	Version history:
	Date        | Version   | Author                    | Remark
	----------------------------------------------------------------------------------------
	 30/03/2023 | 0.1       | R.Golonka                 | First release TIA 17.0 | DHL Munich
	 18/08/2023 | 2.0       | Stefanos Theocharis       | align with Parma UDT
	 06/09/2023 | 2.1       | M.Diebel                  | Reset energy save when NewObjectID is created
	 13/03/2024 | 2.2      | S. Nieswiec                | Added to new baseline

	 *)

	REGION 1 - Chute status move

	    #s_UDT_Downstream_Sorter.Full := #i_UDT_Outfeed2StatesStatus.Specific.ChuteFull;// Downstream sorter status full update

	    #s_UDT_Downstream_Sorter.HalfFull := #i_UDT_Outfeed2StatesStatus.Specific.ChuteHalfFull;   // Downstream sorter status half-full update

	END_REGION

	REGION 2 - Send ready to recevie to crossbelt

	    // Set ready to recevie to Xbelt (when Chute is RTR then XBelt can discharge)
	    #s_UDT_Downstream_Sorter.ReadyToReceive := #iq_UDT_ChuteExternalHandshake.RTR AND (#i_UDT_AssociatedConveyorInterface.VFDatSpeed OR NOT #ix_ConfigHorizontalOutfeed);

	END_REGION

	REGION 3 - Downstream Sorter

	    // Downstream sorter functionality when horizontal outfeed mode is active
	    IF #ix_ConfigHorizontalOutfeed THEN
	        #s_UDT_Downstream_Sorter.Running := #i_UDT_AssociatedConveyorInterface.RunFwd AND NOT #i_UDT_AssociatedConveyorInterface.ManualModeActive;

	    ELSE
	        #s_UDT_Downstream_Sorter.Running := #iq_UDT_ChuteExternalHandshake.RTR; // Downstream sorter functionality when spiral mode is active

	    END_IF;

	END_REGION

	REGION 4 - Package update

	    // Move the current ID to position 0
	    #sa_ExchangeObjectID[0] := #i_UDT_Sorter_Downstream.DischargedObjectID;

	    // When the ID is different with previous ID do:
	    IF #sa_ExchangeObjectID[0] <> #sa_ExchangeObjectID[1] THEN
	        // Update new object
	        #s_UDT_XBeltExitInterface.NewObjectID := TRUE;
	        // Update obejct ID
	        #s_UDT_XBeltExitInterface.ObjectID := #i_UDT_Sorter_Downstream.DischargedObjectID;
	        // Update product lenght
	        #s_UDT_XBeltExitInterface.ProductLength := DINT_TO_INT(#i_UDT_Sorter_Downstream.DischargedPackageLength MOD #c_MaximumLength);
	        // Setting actual value to previous one
	        #sa_ExchangeObjectID[1] := #sa_ExchangeObjectID[0];
	    ELSE
	        #s_UDT_XBeltExitInterface.NewObjectID := FALSE;
	    END_IF;

	    #iq_UDT_ChuteExternalHandshake.RTS := #s_UDT_XBeltExitInterface.NewObjectID;    // Conveyor ready to send if parcel diverted
	    #iq_UDT_ChuteExternalHandshake.ResetEnergySave := #s_UDT_XBeltExitInterface.NewObjectID;
	END_REGION

	REGION 5 - Output update

	    #q_UDT_Downstream_Sorter := #s_UDT_Downstream_Sorter;    // Move UDT Downstream Sorter to output

	    #q_UDT_XBeltExitInterface := #s_UDT_XBeltExitInterface;    // Move Xbelt Exit interface

	END_REGION

	REGION 6 - Status

	    #s_UDT_XBeltExitStatus.ChuteDisabled := #i_UDT_Sorter_Downstream.Basic.ChuteDisabled;   // Status HMI upadate chute disabled

	    #s_UDT_XBeltExitStatus.ChuteJam := #i_UDT_Sorter_Downstream.Basic.ChuteJam;   // Status HMI upadate chute jammed

	    #s_UDT_XBeltExitStatus.ChuteSensorIncongruence := #i_UDT_Sorter_Downstream.Basic.ChuteSensorIncongruence;    // Status HMI update chute sensor incongrunce

	    #q_UDT_XBeltExitStatus := #s_UDT_XBeltExitStatus;  // Move status static to output

	END_REGION


END_FUNCTION_BLOCK

FUNCTION_BLOCK "FB_VFD_MultiControl_Universal_Full"
{ S7_Optimized_Access := 'TRUE' }
AUTHOR : 'KBA-PM'
VERSION : 0.1
// ATTRIBUTES
// AUTO_NUMBER = True
// BLOCK_NUMBER = 106
// END_ATTRIBUTES
   VAR_INPUT
      i_UDT_VFDConfiguration { ExternalAccessible := 'False'; ExternalVisible := 'False'; ExternalWritable := 'False'} : "UDT_VFD_MultiControl_Configuration";   //   VFD configuration structure
      i_UDT_VFDInputs { ExternalAccessible := 'False'; ExternalVisible := 'False'; ExternalWritable := 'False'} : "UDT_VFD_MultiControl_Universal_Full";   //   VFD inputs structure
      ii_MotorNumber { ExternalAccessible := 'False'; ExternalVisible := 'False'; ExternalWritable := 'False'} : Int;   //   Motor number that is connected to the Multicontrol module [1,2,3 or 4]
      ix_PowerOK { ExternalAccessible := 'False'; ExternalVisible := 'False'; ExternalWritable := 'False'} : Bool;   //   TRUE when External Power OK
      ix_SafetyOK { ExternalAccessible := 'False'; ExternalVisible := 'False'; ExternalWritable := 'False'} : Bool;   //   TRUE when Safety OK
      ix_SimulationModeActive { ExternalAccessible := 'False'; ExternalVisible := 'False'; ExternalWritable := 'False'} : Bool;   //   TRUE when Simulation mode active
   END_VAR

   VAR_OUTPUT
      q_UDT_HMIStatus { ExternalAccessible := 'False'; ExternalVisible := 'False'; ExternalWritable := 'False'} : "UDT_VfdStatus";   //   HMI status structure
      qsi_UDT_VFDSpeed { ExternalAccessible := 'False'; ExternalVisible := 'False'; ExternalWritable := 'False'} : SInt;   //   VFD speed setpoint
   END_VAR

   VAR_IN_OUT
      iq_UDT_ConveyorInterface : "UDT_ConveyorInterface";   //   Conveyor interface structure
      iq_UDT_VFDStatistics : "UDT_VfdStatistics";   //   Statistics structure
   END_VAR

   VAR
      s_FB_TimerOnOffDelayCheckSupply { ExternalAccessible := 'False'; ExternalVisible := 'False'; ExternalWritable := 'False'; S7_SetPoint := 'False'} : "FB_TimerOnOffDelay";   //  "TimerOnOffDelay" - to delay time for VFD supply contactor
      s_FB_TimerOnOffDelay_ProfinetNotOnlineMasking { ExternalAccessible := 'False'; ExternalVisible := 'False'; ExternalWritable := 'False'; S7_SetPoint := 'False'} : "FB_TimerOnOffDelay";   //   "TimerOnOffDelay" - to delay time for profinet not online masking
      s_FB_TimerOnOffDelay_ProfinetSlaveErrorMasking { ExternalAccessible := 'False'; ExternalVisible := 'False'; ExternalWritable := 'False'; S7_SetPoint := 'False'} : "FB_TimerOnOffDelay";   //   "TimerOnOffDelay" - to delay time for profinet error masking
      s_FB_TimerOnOffDelay_Instance { ExternalAccessible := 'False'; ExternalVisible := 'False'; ExternalWritable := 'False'; S7_SetPoint := 'False'} : "FB_TimerOnOffDelay";   //   "TimerOnOffDelay" - to delay time for Instance
      s_FB_TimerOnOffDelay_SafetyOK { ExternalAccessible := 'False'; ExternalVisible := 'False'; ExternalWritable := 'False'; S7_SetPoint := 'False'} : "FB_TimerOnOffDelay";   //   "TimerOnOffDelay" - to delay time for safety
      s_FB_TimerOnOffDelay_RunCommand { ExternalAccessible := 'False'; ExternalVisible := 'False'; ExternalWritable := 'False'; S7_SetPoint := 'False'} : "FB_TimerOnOffDelay";   //   "TimerOnOffDelay" - to delay time for run command motor
      s_R_TRIG_RunForward {InstructionName := 'R_TRIG'; LibVersion := '1.0'; ExternalAccessible := 'False'; ExternalVisible := 'False'; ExternalWritable := 'False'; S7_SetPoint := 'False'} : R_TRIG;   //   Rising edge of Run forward signal
      s_R_TRIG_RunReverse {InstructionName := 'R_TRIG'; LibVersion := '1.0'; ExternalAccessible := 'False'; ExternalVisible := 'False'; ExternalWritable := 'False'; S7_SetPoint := 'False'} : R_TRIG;   //   Rising edge of Run reverse
      s_R_TRIG_PNSlaveNotOnline {InstructionName := 'R_TRIG'; LibVersion := '1.0'; ExternalAccessible := 'False'; ExternalVisible := 'False'; ExternalWritable := 'False'; S7_SetPoint := 'False'} : R_TRIG;   //   Rising edge for trigger Profinet slave not online statistics
      s_R_TRIG_PNSlaveError {InstructionName := 'R_TRIG'; LibVersion := '1.0'; ExternalAccessible := 'False'; ExternalVisible := 'False'; ExternalWritable := 'False'; S7_SetPoint := 'False'} : R_TRIG;   //   Rising edge for trigger Profinet slave error statistics
      s_R_TRIG_InternalError {InstructionName := 'R_TRIG'; LibVersion := '1.0'; ExternalAccessible := 'False'; ExternalVisible := 'False'; ExternalWritable := 'False'; S7_SetPoint := 'False'} : R_TRIG;   //   Rising edge for trigger Internal VFD Error statistics
      s_R_TRIG_Running {InstructionName := 'R_TRIG'; LibVersion := '1.0'; ExternalAccessible := 'False'; ExternalVisible := 'False'; ExternalWritable := 'False'; S7_SetPoint := 'False'} : R_TRIG;   //   Rising edge for starting of the running signal
      s_R_TRIG_Instance {InstructionName := 'R_TRIG'; LibVersion := '1.0'; ExternalAccessible := 'False'; ExternalVisible := 'False'; ExternalWritable := 'False'; S7_SetPoint := 'False'} : R_TRIG;   //   Raising edge for Instance
      s_R_TRIG_NewPNSlaveError {InstructionName := 'R_TRIG'; LibVersion := '1.0'; ExternalAccessible := 'False'; ExternalVisible := 'False'; ExternalWritable := 'False'; S7_SetPoint := 'False'} : R_TRIG;   //   New profinet slave error trigger
      s_R_TRIG_NewPNSlaveNotOnline {InstructionName := 'R_TRIG'; LibVersion := '1.0'; ExternalAccessible := 'False'; ExternalVisible := 'False'; ExternalWritable := 'False'; S7_SetPoint := 'False'} : R_TRIG;   //   New profinet slave not online trigger
      s_UDT_HMIStatus { ExternalAccessible := 'False'; ExternalVisible := 'False'; ExternalWritable := 'False'; S7_SetPoint := 'False'} : "UDT_VfdStatus";   //   HMI status structure
      s_UDT_PNDevice { ExternalAccessible := 'False'; ExternalVisible := 'False'; ExternalWritable := 'False'; S7_SetPoint := 'False'} : "UDT_PNDevice";   //   PN device info structure
      ss_VFDGeoStruct {InstructionName := 'GEOADDR'; LibVersion := '1.0'; ExternalAccessible := 'False'; ExternalVisible := 'False'; ExternalWritable := 'False'; S7_SetPoint := 'False'} : GEOADDR;   //   Geo structure indicate to telegram
      ss_RDREC { ExternalAccessible := 'False'; ExternalVisible := 'False'; ExternalWritable := 'False'} : Struct   //   Read error code record structure
         Valid { ExternalAccessible := 'False'; ExternalVisible := 'False'; ExternalWritable := 'False'} : Bool;   //      Read operation is done
         Busy { ExternalAccessible := 'False'; ExternalVisible := 'False'; ExternalWritable := 'False'} : Bool;   //      Read operation is in progress
         Error { ExternalAccessible := 'False'; ExternalVisible := 'False'; ExternalWritable := 'False'} : Bool;   //      Read operation has an error
         Status { ExternalAccessible := 'False'; ExternalVisible := 'False'; ExternalWritable := 'False'} : DWord;   //      Read operation status
         Lenght { ExternalAccessible := 'False'; ExternalVisible := 'False'; ExternalWritable := 'False'} : UInt;   //      Lenght of the read record
      END_STRUCT;
      ss_WRREC { ExternalAccessible := 'False'; ExternalVisible := 'False'; ExternalWritable := 'False'} : Struct   //   Write record structure
         Acceleration { ExternalAccessible := 'False'; ExternalVisible := 'False'; ExternalWritable := 'False'} : Struct   //      Acceleration
            REQ { ExternalAccessible := 'False'; ExternalVisible := 'False'; ExternalWritable := 'False'} : Bool;   //      Requirement
            Index { ExternalAccessible := 'False'; ExternalVisible := 'False'; ExternalWritable := 'False'} : DInt;   //      Index
            Done { ExternalAccessible := 'False'; ExternalVisible := 'False'; ExternalWritable := 'False'} : Bool;   //      Operation is done
            Busy { ExternalAccessible := 'False'; ExternalVisible := 'False'; ExternalWritable := 'False'} : Bool;   //      Write operation is in progress
            Error { ExternalAccessible := 'False'; ExternalVisible := 'False'; ExternalWritable := 'False'} : Bool;   //      Write operation has an error
            Status { ExternalAccessible := 'False'; ExternalVisible := 'False'; ExternalWritable := 'False'} : DWord;   //      Write operation status
            Data { ExternalAccessible := 'False'; ExternalVisible := 'False'; ExternalWritable := 'False'} : Word;   //      Data to write
         END_STRUCT;
         Deceleration { ExternalAccessible := 'False'; ExternalVisible := 'False'; ExternalWritable := 'False'} : Struct   //      Deceleration
            REQ { ExternalAccessible := 'False'; ExternalVisible := 'False'; ExternalWritable := 'False'} : Bool;   //      Requirement
            Index { ExternalAccessible := 'False'; ExternalVisible := 'False'; ExternalWritable := 'False'} : DInt;   //      Index
            Done { ExternalAccessible := 'False'; ExternalVisible := 'False'; ExternalWritable := 'False'} : Bool;   //      Operation is done
            Busy { ExternalAccessible := 'False'; ExternalVisible := 'False'; ExternalWritable := 'False'} : Bool;   //      Write operation is in progress
            Error { ExternalAccessible := 'False'; ExternalVisible := 'False'; ExternalWritable := 'False'} : Bool;   //      Write operation has an error
            Status { ExternalAccessible := 'False'; ExternalVisible := 'False'; ExternalWritable := 'False'} : DWord;   //      Write operation status
            Data { ExternalAccessible := 'False'; ExternalVisible := 'False'; ExternalWritable := 'False'} : Word;   //      Data to write
         END_STRUCT;
      END_STRUCT;
      s_RDREC_ErrorCode {InstructionName := 'RDREC'; LibVersion := '1.0'; ExternalAccessible := 'False'; ExternalVisible := 'False'; ExternalWritable := 'False'; S7_SetPoint := 'False'} : RDREC;   //   Read error code record instruction
      s_WRREC_ACC {InstructionName := 'WRREC'; LibVersion := '1.1'; ExternalAccessible := 'False'; ExternalVisible := 'False'; ExternalWritable := 'False'; S7_SetPoint := 'False'} : WRREC;   //   Write acceleration record inctruction
      s_WRREC_DEC {InstructionName := 'WRREC'; LibVersion := '1.1'; ExternalAccessible := 'False'; ExternalVisible := 'False'; ExternalWritable := 'False'; S7_SetPoint := 'False'} : WRREC;   //   Write deceleration record instruction
      shw_VFD_Telegram { ExternalAccessible := 'False'; ExternalVisible := 'False'; ExternalWritable := 'False'} : HW_ANY;   //   Free telegram's HW_ID
      sr_MaximumSpeed { ExternalAccessible := 'False'; ExternalVisible := 'False'; ExternalWritable := 'False'} : Real;   //   Maximum speed [mm/s]
      sr_SpeedsetpointCorrected { ExternalAccessible := 'False'; ExternalVisible := 'False'; ExternalWritable := 'False'} : Real;   //  Speedsetpoint corrected with factor
      sw_ErrorCode { ExternalAccessible := 'False'; ExternalVisible := 'False'; ExternalWritable := 'False'} : Word;   //   VFD error code
      si_RequiredSpeedSetpoint { ExternalAccessible := 'False'; ExternalVisible := 'False'; ExternalWritable := 'False'} : Int;   //   Required speed setpoint
      si_AccelerationSetpoint { ExternalAccessible := 'False'; ExternalVisible := 'False'; ExternalWritable := 'False'} : Int;   //   Acceleration setpoint value
      si_DecelerationSetpoint { ExternalAccessible := 'False'; ExternalVisible := 'False'; ExternalWritable := 'False'} : Int;   //   Deceleration setpoint value
      si_AccelerationOld { ExternalAccessible := 'False'; ExternalVisible := 'False'; ExternalWritable := 'False'} : Int;   //   Old acceleration value
      si_DecelerationOld { ExternalAccessible := 'False'; ExternalVisible := 'False'; ExternalWritable := 'False'} : Int;   //   Old deceleration value
      si_ActualSpeed { ExternalAccessible := 'False'; ExternalVisible := 'False'; ExternalWritable := 'False'} : Int;   //   Actual speed in [mm/s]
      si_Log2GeoReturn { ExternalAccessible := 'False'; ExternalVisible := 'False'; ExternalWritable := 'False'} : Int;   //   Log2Geo function return
      si_Geo2LogReturn { ExternalAccessible := 'False'; ExternalVisible := 'False'; ExternalWritable := 'False'} : Int;   //   Geo2Log function return
      sx_PNSlaveErrorCount { ExternalAccessible := 'False'; ExternalVisible := 'False'; ExternalWritable := 'False'} : Int;   //   Profinet slave error counter
      sx_PNSlaveNotOnlineCount { ExternalAccessible := 'False'; ExternalVisible := 'False'; ExternalWritable := 'False'} : Int;   //   Profinet slave not online counter
      ssi_MotorSpeed { ExternalAccessible := 'False'; ExternalVisible := 'False'; ExternalWritable := 'False'} : SInt;   //   Motor speed value
      sx_ConfigurationError { ExternalAccessible := 'False'; ExternalVisible := 'False'; ExternalWritable := 'False'} : Bool;   //   Commissioning: configuration error
      sx_PNDeviceHealthy { ExternalAccessible := 'False'; ExternalVisible := 'False'; ExternalWritable := 'False'} : Bool;   //   Profinet device is online and error free
      sx_PowerOk { ExternalAccessible := 'False'; ExternalVisible := 'False'; ExternalWritable := 'False'} : Bool;   //   Communication, safety and power are available
      sx_VFD_Available { ExternalAccessible := 'False'; ExternalVisible := 'False'; ExternalWritable := 'False'} : Bool;   //   Hardware of VFD is ok
      sx_ErrorActive { ExternalAccessible := 'False'; ExternalVisible := 'False'; ExternalWritable := 'False'} : Bool;   //   Block has an error
      sx_InvalidMotorNumber { ExternalAccessible := 'False'; ExternalVisible := 'False'; ExternalWritable := 'False'} : Bool;   //   Invalid motor error
      sx_MotorError { ExternalAccessible := 'False'; ExternalVisible := 'False'; ExternalWritable := 'False'} : Bool;   //   Motor error
      sx_EnableOperation { ExternalAccessible := 'False'; ExternalVisible := 'False'; ExternalWritable := 'False'} : Bool;   //   Enable operation signal
      sx_RunVFDForward { ExternalAccessible := 'False'; ExternalVisible := 'False'; ExternalWritable := 'False'} : Bool;   //   Start VFD forward
      sx_RunVFDReverse { ExternalAccessible := 'False'; ExternalVisible := 'False'; ExternalWritable := 'False'} : Bool;   //   Start VFD backward
      sx_AccelerationDone { ExternalAccessible := 'False'; ExternalVisible := 'False'; ExternalWritable := 'False'} : Bool;   //   Acceleration is written
      sx_DecelerationDone { ExternalAccessible := 'False'; ExternalVisible := 'False'; ExternalWritable := 'False'} : Bool;   //   Deceleration is written
      sx_SpeedSetpointReached { ExternalAccessible := 'False'; ExternalVisible := 'False'; ExternalWritable := 'False'} : Bool;   //   Motor is running at requested speed
      sx_ErrorDone { ExternalAccessible := 'False'; ExternalVisible := 'False'; ExternalWritable := 'False'} : Bool;   //   Error code is read
      sx_SafetyOK { ExternalAccessible := 'False'; ExternalVisible := 'False'; ExternalWritable := 'False'} : Bool;   //   Safety ok
      sx_MaskingReset { ExternalAccessible := 'False'; ExternalVisible := 'False'; ExternalWritable := 'False'} : Bool;   //   Masking reset
      sx_PNSlaveError { ExternalAccessible := 'False'; ExternalVisible := 'False'; ExternalWritable := 'False'} : Bool;   //   Profinet slave error
      sx_PNSlaveNotOnline { ExternalAccessible := 'False'; ExternalVisible := 'False'; ExternalWritable := 'False'} : Bool;   //   Profinet slave not online
      s_R_TRIG_PNSlaveNotOnline_Acyclic {InstructionName := 'R_TRIG'; LibVersion := '1.0'; ExternalAccessible := 'False'; ExternalVisible := 'False'; ExternalWritable := 'False'; S7_SetPoint := 'False'} : R_TRIG;
   END_VAR

   VAR CONSTANT
      ci_VFDArea : UInt := 1;   //   Area ID of IO Profinet devices
      ci_SubmoduleHWType : UInt := 5;   //   Submodule HW_type number
      ci_TelegramSlot : UInt := 2;   //   Free Siemens telegram slot
      ci_TelegramSubslot : UInt := 1;   //   Free Siemens telegram subslot
      cdi_ErrorCodeIndex : DInt := 17154;   //   Error code index
      cdi_AccelerationIndex : DInt := 18200;   //   Acceleration index
      cdi_DecelerationIndex : DInt := 18204;   //   Deceleration index
   END_VAR


BEGIN
	(*
	----------------------------------------------------------------------------------------
	|                                                                                      |
	|  Copyright  2023             FORTNA Europe BV                                        |
	|  All Rights Reserved         Netherlands                                             |
	|                                                                                      |
	----------------------------------------------------------------------------------------

	Version history:
	Date        | Version   | Author        | Remark
	----------------------------------------------------------------------------------------
	08/11/2019  | 3.0       | A. Nowak      | Initial version
	18/03/2020  | 3.1       | K.Pokorski    | Adapting reviews
	10/06/2021  | 3.2       | L.Klar        | Region 9.1 - #ssi_MotorSpeed = 0 condition commented
	17/11/2021  | 3.3       | P.Gryszczyk   | Region 2 - RunCommand timer changed conditions
	18/02/2021  | 3.4       | P.Gryszczyk   | Region 4 - PNNotOnline and PNSlaveError masking, sending reset to system
	24/05/2023  | 3.5       | S.Nikodem     | Update to DHL Munich specification
	04/07/2023  | 3.7       | P.Gryszczyk   | Changed the PNSlaveNotOnline to R_TRIG for the acyclic writing logic
	13/03/2024  | 4.1       | S. Nieswiec   | Added to new baseline
	*)

	REGION 1 - Get Device Profinet number

	    // Getting information about Profinet Device.
	    "FC_GetDevicePN"(is_PNDeviceName := #i_UDT_VFDConfiguration.VFDPNDeviceName,
	                     ix_SimulationModeActive := #ix_SimulationModeActive,
	                     iqUDT_PND := #s_UDT_PNDevice);

	END_REGION

	REGION 2 - Motor number validation

	    // Check the motor number and copy the it's error status and speed.
	    CASE (#ii_MotorNumber)
	    OF
	        1:
	            // Delay
	            #s_FB_TimerOnOffDelay_RunCommand(iudi_OnDelayTime := 1500,
	                                             ix_SignalToDelay :=
	                                             (#sx_RunVFDForward
	                                             OR #sx_RunVFDReverse)
	                                             AND #i_UDT_VFDInputs.CurrentMotor1 < #i_UDT_VFDConfiguration.MinimumCurrentWhenRunninng);

	            #ssi_MotorSpeed := #i_UDT_VFDInputs.SpeedMotor1;

	            IF (#s_FB_TimerOnOffDelay_RunCommand.qx_DelayedSignal AND #sx_EnableOperation) OR #i_UDT_VFDInputs.ErrorMotor1
	            THEN

	                #sx_MotorError := TRUE;

	            END_IF;
	        2:
	            #s_FB_TimerOnOffDelay_RunCommand(iudi_OnDelayTime := 1500,
	                                             ix_SignalToDelay :=
	                                             (#sx_RunVFDForward
	                                             OR #sx_RunVFDReverse)
	                                             AND #i_UDT_VFDInputs.CurrentMotor2 < #i_UDT_VFDConfiguration.MinimumCurrentWhenRunninng);

	            #ssi_MotorSpeed := #i_UDT_VFDInputs.SpeedMotor2;

	            IF (#s_FB_TimerOnOffDelay_RunCommand.qx_DelayedSignal AND #sx_EnableOperation) OR #i_UDT_VFDInputs.ErrorMotor2

	            THEN

	                #sx_MotorError := TRUE;

	            END_IF;
	        3:
	            #s_FB_TimerOnOffDelay_RunCommand(iudi_OnDelayTime := 1500,
	                                             ix_SignalToDelay :=
	                                             (#sx_RunVFDForward
	                                             OR #sx_RunVFDReverse)
	                                             AND #i_UDT_VFDInputs.CurrentMotor3 < #i_UDT_VFDConfiguration.MinimumCurrentWhenRunninng);

	            #ssi_MotorSpeed := #i_UDT_VFDInputs.SpeedMotor3;

	            IF (#s_FB_TimerOnOffDelay_RunCommand.qx_DelayedSignal AND #sx_EnableOperation) OR #i_UDT_VFDInputs.ErrorMotor3
	            THEN

	                #sx_MotorError := TRUE;

	            END_IF;
	        4:
	            #s_FB_TimerOnOffDelay_RunCommand(iudi_OnDelayTime := 1500,
	                                             ix_SignalToDelay :=
	                                             (#sx_RunVFDForward
	                                             OR #sx_RunVFDReverse)
	                                             AND #i_UDT_VFDInputs.CurrentMotor4 < #i_UDT_VFDConfiguration.MinimumCurrentWhenRunninng);

	            #ssi_MotorSpeed := #i_UDT_VFDInputs.SpeedMotor4;

	            IF (#s_FB_TimerOnOffDelay_RunCommand.qx_DelayedSignal AND #sx_EnableOperation) OR #i_UDT_VFDInputs.ErrorMotor4
	            THEN

	                #sx_MotorError := TRUE;

	            END_IF;

	        ELSE
	            #sx_InvalidMotorNumber := TRUE;
	    END_CASE;

	END_REGION

	REGION 3 - Reset errors

	    // Reset the errors on the command from the conveyor interface.
	    //
	    #s_R_TRIG_Instance(CLK := #ix_SafetyOK,
	                       Q => #sx_SafetyOK);

	    #s_FB_TimerOnOffDelay_Instance(iudi_OffDelayTime := 10000,
	                                   ix_SignalToDelay := #sx_SafetyOK,
	                                   qx_DelayedSignal => #sx_MaskingReset);


	    IF #iq_UDT_ConveyorInterface.InternalErrorReset THEN
	        #s_UDT_HMIStatus.PNSlaveNotonline := FALSE;
	        #s_UDT_HMIStatus.PNSlaveError := FALSE;
	        #s_UDT_HMIStatus.InternalError := FALSE;
	        #sx_InvalidMotorNumber := FALSE;
	        #sx_MotorError := FALSE;
	    END_IF;

	END_REGION

	REGION 4 - Hardware check

	    // Hardware will be available only after the delay, so the device has time for the initialization.
	    #s_FB_TimerOnOffDelayCheckSupply(iudi_OnDelayTime := 2000,
	                                     ix_SignalToDelay := #ix_PowerOK,
	                                     qx_DelayedSignal => #sx_PowerOk);

	    #s_FB_TimerOnOffDelay_ProfinetNotOnlineMasking(iudi_OnDelayTime := #i_UDT_VFDConfiguration.TimePNErrorMasking,
	                                                   iudi_OffDelayTime := 0,
	                                                   ix_SignalToDelay := #sx_PNSlaveNotOnline,
	                                                   qx_DelayedSignal => #s_UDT_HMIStatus.PNSlaveNotonline);

	    #s_FB_TimerOnOffDelay_ProfinetSlaveErrorMasking(iudi_OnDelayTime := #i_UDT_VFDConfiguration.TimePNErrorMasking,
	                                                    iudi_OffDelayTime := 0,
	                                                    ix_SignalToDelay := #sx_PNSlaveError,
	                                                    qx_DelayedSignal => #s_UDT_HMIStatus.PNSlaveError);

	    #s_R_TRIG_NewPNSlaveNotOnline(CLK := #sx_PNSlaveNotOnline);
	    #s_R_TRIG_NewPNSlaveError(CLK := #sx_PNSlaveError);
	    // Check if PN device is online.
	    IF NOT "DB_ProfinetDiagnostic".ProfinetNetworks[#s_UDT_PNDevice.PNNetworknumber].DeviceStatus[#s_UDT_PNDevice.PNDeviceNumber].DeviceState.Exist
	        AND NOT #ix_SimulationModeActive
	        AND #sx_PowerOk
	    THEN
	        #sx_PNSlaveNotOnline := TRUE;
	    ELSE
	        #sx_PNSlaveNotOnline := FALSE;
	    END_IF;

	    IF #s_R_TRIG_NewPNSlaveNotOnline.Q THEN
	        #sx_PNSlaveNotOnlineCount += 1;
	    END_IF;

	    // Check if PN device has an error.
	    IF "DB_ProfinetDiagnostic".ProfinetNetworks[#s_UDT_PNDevice.PNNetworknumber].DeviceStatus[#s_UDT_PNDevice.PNDeviceNumber].DeviceState.Error
	        AND NOT #ix_SimulationModeActive
	        AND #sx_PowerOk
	    THEN
	        #sx_PNSlaveError := TRUE;
	    ELSE
	        #sx_PNSlaveError := FALSE;
	    END_IF;

	    IF #s_R_TRIG_NewPNSlaveError.Q THEN
	        #sx_PNSlaveErrorCount += 1;
	    END_IF;

	    // Set bit when PN device is healthy (online and no error).
	    #sx_PNDeviceHealthy :=
	    NOT #s_UDT_HMIStatus.PNSlaveNotonline
	    AND NOT #s_UDT_HMIStatus.PNSlaveError
	    AND #s_UDT_PNDevice.PNDeviceFound
	    AND #sx_PowerOk;

	    // Set VFD available bit when all conditions are met.
	    #sx_VFD_Available :=
	    (NOT #sx_MotorError
	    AND #sx_PowerOk
	    AND #sx_PNDeviceHealthy)
	    OR #ix_SimulationModeActive;

	END_REGION

	REGION 5 - Extract telegram's HW_ID

	    // Extract telegram's HW_ID
	    #si_Log2GeoReturn := LOG2GEO(LADDR := "DB_ProfinetDiagnostic".ProfinetNetworks[#s_UDT_PNDevice.PNNetworknumber].DeviceStatus[#s_UDT_PNDevice.PNDeviceNumber].DeviceState.HW_ID, GEOADDR := #ss_VFDGeoStruct);
	    #ss_VFDGeoStruct.AREA := #ci_VFDArea;
	    #ss_VFDGeoStruct.HWTYPE := #ci_SubmoduleHWType;
	    #ss_VFDGeoStruct.STATION := INT_TO_UINT(#s_UDT_PNDevice.PNDeviceNumber);
	    #ss_VFDGeoStruct.SLOT := #ci_TelegramSlot;
	    #ss_VFDGeoStruct.SUBSLOT := #ci_TelegramSubslot;

	    #si_Geo2LogReturn := GEO2LOG(GEOADDR := #ss_VFDGeoStruct, LADDR => #shw_VFD_Telegram);

	END_REGION

	REGION 6 - Check errors

	    #s_FB_TimerOnOffDelay_SafetyOK(iudi_OnDelayTime := 10000,
	                                   ix_SignalToDelay := #ix_SafetyOK);

	    // Check if the motor has an error.
	    IF #s_FB_TimerOnOffDelay_SafetyOK.qx_DelayedSignal  //#ix_SafetyOK
	    THEN
	        #s_UDT_HMIStatus.InternalError := #sx_MotorError;

	    END_IF;
	    // Create trigger on error.
	    #s_R_TRIG_InternalError(CLK := #s_UDT_HMIStatus.InternalError);

	    // If the internal error occured, reset the error code read done signal.
	    IF #s_R_TRIG_InternalError.Q
	    THEN
	        #sx_ErrorDone := FALSE;
	    END_IF;

	    // If there is an internal error, read the error code from the Interroll VFD. Otherwise, reset it.
	    IF NOT #s_UDT_HMIStatus.InternalError
	    THEN
	        #s_UDT_HMIStatus.ErrorCode := 0;
	    ELSE
	        // Read the error code from the multicontrol.
	        #s_RDREC_ErrorCode(REQ := ((NOT #sx_ErrorDone OR "mx_FirstScan") AND NOT #s_UDT_HMIStatus.PNSlaveNotonline),
	                           ID := #shw_VFD_Telegram,
	                           INDEX := #cdi_ErrorCodeIndex,
	                           MLEN := 0,
	                           VALID => #ss_RDREC.Valid,
	                           BUSY => #ss_RDREC.Busy,
	                           ERROR => #ss_RDREC.Error,
	                           STATUS => #ss_RDREC.Status,
	                           LEN => #ss_RDREC.Lenght,
	                           RECORD := #sw_ErrorCode);

	        // IF error code is read, set the error code read signal and write it to the structure.
	        IF #s_RDREC_ErrorCode.VALID
	        THEN
	            #sx_ErrorDone := TRUE;
	            #s_UDT_HMIStatus.ErrorCode := WORD_TO_INT(SWAP_WORD(IN := #sw_ErrorCode));
	        END_IF;
	    END_IF;

	END_REGION

	REGION 7 - Check if configuration is ok for commissioning purposes

	    // Validate the VFD configuration and motor number.
	    IF #i_UDT_VFDConfiguration.MaximumSpeed > 0.0
	        AND #i_UDT_VFDConfiguration.VFDRampUpTime > 0
	        AND #i_UDT_VFDConfiguration.VFDRampDownTime > 0
	        AND NOT #sx_InvalidMotorNumber
	    THEN
	        #sx_ConfigurationError := FALSE;
	    ELSE
	        #sx_ConfigurationError := TRUE;
	    END_IF;

	END_REGION

	REGION 8 - Handle speed

	    // Write max speed to static.
	    #sr_MaximumSpeed := #i_UDT_VFDConfiguration.MaximumSpeed;

	    // Use correction factor to calculate setpint for diaginal use
	    #sr_SpeedsetpointCorrected := INT_TO_REAL(#iq_UDT_ConveyorInterface.SpeedSetpoint) * #i_UDT_VFDConfiguration.CorrectionFactor;

	    // Actual speed setpoint
	    #si_RequiredSpeedSetpoint := REAL_TO_INT((#sr_SpeedsetpointCorrected * 100.0) / (#sr_MaximumSpeed));

	    // Speed setpoint saturation in case when the speed setpoint is higher than the max speed.
	    IF #si_RequiredSpeedSetpoint > 100
	    THEN
	        #si_RequiredSpeedSetpoint := 100;
	        #iq_UDT_ConveyorInterface.ConfigurationError := TRUE;
	    ELSIF #si_RequiredSpeedSetpoint < -100
	    THEN
	        #si_RequiredSpeedSetpoint := -100;
	        #iq_UDT_ConveyorInterface.ConfigurationError := TRUE;
	    END_IF;
	END_REGION

	REGION 9 - Prepare output data VFD

	    REGION 9.1 - Set speed setpoint in forward and reverse direction
	        // Get rising edge of Run forward and reverse signal.
	        #s_R_TRIG_RunForward(CLK := #iq_UDT_ConveyorInterface.RunFwd);
	        #s_R_TRIG_RunReverse(CLK := #iq_UDT_ConveyorInterface.RunRvs);

	        // When rising edge of the forward or reverse signal is received, the drive has to stop to be able to make the switch.
	        IF #s_R_TRIG_RunForward.Q
	            OR #s_R_TRIG_RunReverse.Q
	        THEN
	            #qsi_UDT_VFDSpeed := 0;
	        END_IF;

	        // If motor stopped and Run forward is requested and forward direction is interlock, set run forward signal and reset run reverse signal.
	        IF //#ssi_MotorSpeed = 0 and
	            #iq_UDT_ConveyorInterface.RunFwd
	            AND #i_UDT_VFDConfiguration.InterlockFwd
	        THEN
	            #sx_RunVFDForward := TRUE;
	            #sx_RunVFDReverse := FALSE;
	        END_IF;

	        // If motor stopped and Run reverse is requested and reverse direction is interlock, set run reverse signal and reset run forward signal.
	        IF // #ssi_MotorSpeed = 0 AND
	            #iq_UDT_ConveyorInterface.RunRvs
	            AND #i_UDT_VFDConfiguration.InterlockRvs
	        THEN
	            #sx_RunVFDReverse := TRUE;
	            #sx_RunVFDForward := FALSE;
	        END_IF;

	    END_REGION

	    REGION 9.2 - Stopping

	        // Stop the VFD if one of the following conditions is met.
	        IF (NOT #iq_UDT_ConveyorInterface.RunRvs AND NOT #iq_UDT_ConveyorInterface.RunFwd)
	            OR (#iq_UDT_ConveyorInterface.RunRvs AND #iq_UDT_ConveyorInterface.RunFwd)
	            OR (#sx_RunVFDReverse AND NOT #i_UDT_VFDConfiguration.InterlockRvs)
	            OR (#sx_RunVFDForward AND NOT #i_UDT_VFDConfiguration.InterlockFwd)
	            OR ((#s_R_TRIG_RunForward.Q AND #ssi_MotorSpeed < 0)
	            OR (#s_R_TRIG_RunReverse.Q AND #ssi_MotorSpeed > 0))
	        THEN
	            #sx_RunVFDReverse := FALSE;
	            #sx_RunVFDForward := FALSE;
	        END_IF;

	    END_REGION

	    REGION 9.3 - Check for enable operation signal

	        // Operation is enable when VFD is available and there is one of the run commands.
	        #sx_EnableOperation :=
	        #sx_VFD_Available
	        AND (#sx_RunVFDForward OR #sx_RunVFDReverse)
	        AND NOT #sx_ConfigurationError;

	    END_REGION

	END_REGION

	REGION 10 - Write outputs to VFD

	    REGION 10.1 - Write speed setpoint to drive

	        // The conveyor stopped and may now run in forward direction.
	        IF ((#sx_RunVFDForward AND NOT #i_UDT_VFDConfiguration.DirectionReversal)
	            OR (#sx_RunVFDReverse AND #i_UDT_VFDConfiguration.DirectionReversal))
	            AND #sx_EnableOperation
	        THEN
	            #qsi_UDT_VFDSpeed := INT_TO_SINT(#si_RequiredSpeedSetpoint);
	        END_IF;

	        // The conveyor stopped and may now run in reverse direction.
	        IF ((#sx_RunVFDReverse AND NOT #i_UDT_VFDConfiguration.DirectionReversal)
	            OR (#sx_RunVFDForward AND #i_UDT_VFDConfiguration.DirectionReversal))
	            AND #sx_EnableOperation
	        THEN
	            #qsi_UDT_VFDSpeed := - INT_TO_SINT(#si_RequiredSpeedSetpoint);
	        END_IF;

	        // Clear speed setpoint when run isn't request.
	        IF (NOT #sx_RunVFDForward
	            AND NOT #sx_RunVFDReverse)
	            OR NOT #sx_EnableOperation
	        THEN
	            #qsi_UDT_VFDSpeed := 0;
	        END_IF;

	    END_REGION

	    REGION 10.2 - Calculate acceleration and deceleration values

	        // Recalculating Acceleration ramp - deviding maximum configured speed by Ramp up time and devide it by 1000.
	        #si_AccelerationSetpoint := REAL_TO_INT(#sr_MaximumSpeed / (UDINT_TO_REAL(#i_UDT_VFDConfiguration.VFDRampUpTime) / 1000.0));

	        // Recalculating Deceleration ramp - deviding maximum configured speed by Ramp down time and devide it by 1000.
	        #si_DecelerationSetpoint := REAL_TO_INT(#sr_MaximumSpeed / (UDINT_TO_REAL(#i_UDT_VFDConfiguration.VFDRampDownTime) / 1000.0));

	    END_REGION

	    REGION 10.3 - Write acceleration to drive

	        #s_R_TRIG_PNSlaveNotOnline_Acyclic(CLK := NOT #s_UDT_HMIStatus.PNSlaveNotonline);

	        // Acceleration write operation is done.
	        IF #sx_AccelerationDone
	        THEN
	            // There is new acceleration value or device is offline.
	            IF #si_AccelerationSetpoint <> #si_AccelerationOld
	                OR #s_R_TRIG_PNSlaveNotOnline_Acyclic.Q
	            THEN
	                // Reset the accleration operation done signal.
	                #sx_AccelerationDone := FALSE;
	            END_IF;
	        END_IF;

	        // The acceleration operation isn't done or there is first scan and device is online.
	        IF (NOT #sx_AccelerationDone OR "mx_FirstScan")
	            AND NOT #s_UDT_HMIStatus.PNSlaveNotonline
	        THEN
	            // There isn't an invalid motor number error and acceleration isn't equal to 0.
	            IF NOT #sx_InvalidMotorNumber
	                AND #si_AccelerationSetpoint > 0
	            THEN
	                // Calculate the index of the acceleration.
	                #ss_WRREC.Acceleration.Index := #cdi_AccelerationIndex + #ii_MotorNumber;
	                // Prepare the data.
	                #ss_WRREC.Acceleration.Data := SWAP(INT_TO_WORD(#si_AccelerationSetpoint));
	                // Set operation is required.
	                #ss_WRREC.Acceleration.REQ := TRUE;

	                // Send acceleration to the device.
	                #s_WRREC_ACC(REQ := #ss_WRREC.Acceleration.REQ,
	                             ID := #shw_VFD_Telegram,
	                             INDEX := #ss_WRREC.Acceleration.Index,
	                             LEN := 0,
	                             DONE => #ss_WRREC.Acceleration.Done,
	                             BUSY => #ss_WRREC.Acceleration.Busy,
	                             ERROR => #ss_WRREC.Acceleration.Error,
	                             STATUS => #ss_WRREC.Acceleration.Status,
	                             RECORD := #ss_WRREC.Acceleration.Data);

	                // Send operation is done.
	                IF #ss_WRREC.Acceleration.Done
	                THEN
	                    // Reset operation is required bit.
	                    #ss_WRREC.Acceleration.REQ := FALSE;
	                    // Set the operation is done signal.
	                    #sx_AccelerationDone := TRUE;
	                    // Write acceleration value into the old one.
	                    #si_AccelerationOld := #si_AccelerationSetpoint;
	                END_IF;
	            END_IF;
	        END_IF;

	    END_REGION

	    REGION 10.4 - Write deceleration to drive

	        // Deceleration write operation is done.
	        IF #sx_DecelerationDone
	        THEN
	            // There is new deceleration value or device is offline.
	            IF #si_DecelerationSetpoint <> #si_DecelerationOld
	                OR #s_R_TRIG_PNSlaveNotOnline_Acyclic.Q
	            THEN
	                // Reset the deceleration operation done signal.
	                #sx_DecelerationDone := FALSE;
	            END_IF;
	        END_IF;

	        // The deceleration operation isn't done or there is first scan and device is online.
	        IF (NOT #sx_DecelerationDone OR "mx_FirstScan")
	            AND NOT #s_UDT_HMIStatus.PNSlaveNotonline
	        THEN
	            // There isn't an invalid motor number error and deceleration isn't equal to 0.
	            IF NOT #sx_InvalidMotorNumber
	                AND #si_DecelerationSetpoint > 0
	            THEN
	                // Calculate the index of the deceleration.
	                #ss_WRREC.Deceleration.Index := #cdi_DecelerationIndex + #ii_MotorNumber;
	                // Prepare the data.
	                #ss_WRREC.Deceleration.Data := SWAP(INT_TO_WORD(#si_DecelerationSetpoint));
	                // Set operation is required.
	                #ss_WRREC.Deceleration.REQ := TRUE;

	                // Send deceleration to the device.
	                #s_WRREC_DEC(REQ := #ss_WRREC.Deceleration.REQ,
	                             ID := #shw_VFD_Telegram,
	                             INDEX := #ss_WRREC.Deceleration.Index,
	                             LEN := 0,
	                             DONE => #ss_WRREC.Deceleration.Done,
	                             BUSY => #ss_WRREC.Deceleration.Busy,
	                             ERROR => #ss_WRREC.Deceleration.Error,
	                             STATUS => #ss_WRREC.Deceleration.Status,
	                             RECORD := #ss_WRREC.Deceleration.Data);

	                // Send operation is done.
	                IF #ss_WRREC.Deceleration.Done
	                THEN
	                    // Reset operation is required bit.
	                    #ss_WRREC.Deceleration.REQ := FALSE;
	                    // Set the operation is done signal.
	                    #sx_DecelerationDone := TRUE;
	                    // Write deceleration value into the old one.
	                    #si_DecelerationOld := #si_DecelerationSetpoint;
	                END_IF;
	            END_IF;
	        END_IF;

	    END_REGION

	END_REGION

	REGION 11 - Copy signals to interface DB and to status output UDT

	    // Create collective error.
	    #sx_ErrorActive :=
	    #s_UDT_HMIStatus.PNSlaveNotonline
	    OR #s_UDT_HMIStatus.PNSlaveError
	    OR #s_UDT_HMIStatus.InternalError
	    OR #sx_ConfigurationError;

	    // Motor is giving direct signal on start, move setpoint to actual speed.
	    IF #ssi_MotorSpeed <> 0
	    THEN
	        #si_ActualSpeed := #iq_UDT_ConveyorInterface.SpeedSetpoint;
	        #sx_SpeedSetpointReached := TRUE;
	    ELSE
	        #si_ActualSpeed := 0;
	        #sx_SpeedSetpointReached := FALSE;
	    END_IF;

	    // Write interface bits.
	    #iq_UDT_ConveyorInterface.VFDRunning :=
	    #sx_VFD_Available
	    AND #iq_UDT_ConveyorInterface.ActualSpeed <> 0;

	    // Speed setpoint is reached.
	    #iq_UDT_ConveyorInterface.VFDatSpeed :=
	    #sx_SpeedSetpointReached
	    AND #sx_VFD_Available;

	    // Set the internal VFD error bit if any fault is active.
	    #iq_UDT_ConveyorInterface.InternalErrorVFD := #sx_ErrorActive;
	    // Copy the speed value to the output.
	    #iq_UDT_ConveyorInterface.ActualSpeed := #si_ActualSpeed;

	    // Copy error status to output.
	    #q_UDT_HMIStatus := #s_UDT_HMIStatus;

	END_REGION

	REGION 12 - Statistics

	    // Create trigger on error and create statistics for profinet slave not online.
	    #s_R_TRIG_PNSlaveNotOnline(CLK := #s_UDT_HMIStatus.PNSlaveNotonline);

	    IF #iq_UDT_ConveyorInterface.ResetStatistics
	        OR #s_UDT_HMIStatus.PNSlaveNotonline
	    THEN
	        "FC_Statistics"(ix_Reset := #iq_UDT_ConveyorInterface.ResetStatistics,
	                        ix_Activate := #s_UDT_HMIStatus.PNSlaveNotonline,
	                        ix_RTrigActivate := #s_R_TRIG_PNSlaveNotOnline.Q,
	                        iqUDT_Statistics := #iq_UDT_VFDStatistics.PNSlaveNotOnline);
	    END_IF;

	    // Create trigger on error and create statistics for profinet slave error.
	    #s_R_TRIG_PNSlaveError(CLK := #s_UDT_HMIStatus.PNSlaveError);

	    IF #iq_UDT_ConveyorInterface.ResetStatistics
	        OR #s_UDT_HMIStatus.PNSlaveError
	    THEN
	        "FC_Statistics"(ix_Reset := #iq_UDT_ConveyorInterface.ResetStatistics,
	                        ix_Activate := #s_UDT_HMIStatus.PNSlaveError,
	                        ix_RTrigActivate := #s_R_TRIG_PNSlaveError.Q,
	                        iqUDT_Statistics := #iq_UDT_VFDStatistics.PNSlaveError);
	    END_IF;

	    IF #iq_UDT_ConveyorInterface.ResetStatistics
	        OR #s_UDT_HMIStatus.InternalError
	    THEN
	        "FC_Statistics"(ix_Reset := #iq_UDT_ConveyorInterface.ResetStatistics,
	                        ix_Activate := #s_UDT_HMIStatus.InternalError,
	                        ix_RTrigActivate := #s_R_TRIG_InternalError.Q,
	                        iqUDT_Statistics := #iq_UDT_VFDStatistics.VFDInternalError);
	    END_IF;

	    // Create trigger on running signal and create statistics for running status.
	    #s_R_TRIG_Running(CLK := #iq_UDT_ConveyorInterface.VFDRunning);

	    IF #iq_UDT_ConveyorInterface.ResetStatistics
	        OR #iq_UDT_ConveyorInterface.VFDRunning
	    THEN
	        "FC_Statistics"(ix_Reset := #iq_UDT_ConveyorInterface.ResetStatistics,
	                        ix_Activate := #iq_UDT_ConveyorInterface.VFDRunning,
	                        ix_RTrigActivate := #s_R_TRIG_Running.Q,
	                        iqUDT_Statistics := #iq_UDT_VFDStatistics.Running);
	    END_IF;

	END_REGION
END_FUNCTION_BLOCK

FUNCTION_BLOCK "FB_Xray_SerialCommunication_Send"
{ S7_Optimized_Access := 'TRUE' }
VERSION : 0.1
// ATTRIBUTES
// AUTO_NUMBER = True
// BLOCK_NUMBER = 113
// END_ATTRIBUTES
   VAR_INPUT
      i_UDT_SerialCommunicationConfiguration { ExternalAccessible := 'False'; ExternalVisible := 'False'; ExternalWritable := 'False'} : "UDT_SerialComConfiguration";   // Serial communication configuration
      is_ActualTime { ExternalAccessible := 'False'; ExternalVisible := 'False'; ExternalWritable := 'False'} : String;   // Actual date and time in String
      ix_EnableSend { ExternalAccessible := 'False'; ExternalVisible := 'False'; ExternalWritable := 'False'} : Bool;   // Enable send
   END_VAR

   VAR_OUTPUT
      q_UDT_Status { ExternalAccessible := 'False'; ExternalVisible := 'False'; ExternalWritable := 'False'} : "UDT_SerialCommunicationSendStatus";   // Status structure
   END_VAR

   VAR_IN_OUT
      iq_UDT_XrayInterface : "UDT_XrayInterface";   // Xray interface structure
   END_VAR

   VAR
      s_Send_P2P {InstructionName := 'Send_P2P'; LibVersion := '4.0'; ExternalAccessible := 'False'; ExternalVisible := 'False'; ExternalWritable := 'False'; S7_SetPoint := 'False'} : Send_P2P;   // PtP send standard function
      s_UDT_Status { ExternalAccessible := 'False'; ExternalVisible := 'False'; ExternalWritable := 'False'; S7_SetPoint := 'False'} : "UDT_SerialCommunicationSendStatus";   // Status structure
      ss_MessageBuffer { ExternalAccessible := 'False'; ExternalVisible := 'False'; ExternalWritable := 'False'} : Struct   // Message stucture
         PieceID { ExternalAccessible := 'False'; ExternalVisible := 'False'; ExternalWritable := 'False'} : String[40];   // Piece ID
         VID { ExternalAccessible := 'False'; ExternalVisible := 'False'; ExternalWritable := 'False'} : String[16];   // VID
         RoutingCode { ExternalAccessible := 'False'; ExternalVisible := 'False'; ExternalWritable := 'False'} : String[2];   // Routing Code
      END_STRUCT;
      ss_Counter { ExternalAccessible := 'False'; ExternalVisible := 'False'; ExternalWritable := 'False'} : Struct   // Counterts only for statistics
         SendMessage { ExternalAccessible := 'False'; ExternalVisible := 'False'; ExternalWritable := 'False'} : UDInt;   // Counter of send message requests
         MessageSent { ExternalAccessible := 'False'; ExternalVisible := 'False'; ExternalWritable := 'False'} : UDInt;   // Counter of correct sent messages
         WrongMessageLength { ExternalAccessible := 'False'; ExternalVisible := 'False'; ExternalWritable := 'False'} : UDInt;   // Counter of a prepared messages with wrong length
         MessageNotSent { ExternalAccessible := 'False'; ExternalVisible := 'False'; ExternalWritable := 'False'} : UDInt;   // Counter of not sent messages
      END_STRUCT;
      ss_Message { ExternalAccessible := 'False'; ExternalVisible := 'False'; ExternalWritable := 'False'} : String;   // Prepared message
      si_OldGIN { ExternalAccessible := 'False'; ExternalVisible := 'False'; ExternalWritable := 'False'} : Int;   // Old GIN number
      si_GIN { ExternalAccessible := 'False'; ExternalVisible := 'False'; ExternalWritable := 'False'} : Int;   // GIN number
      sx_SendMessage { ExternalAccessible := 'False'; ExternalVisible := 'False'; ExternalWritable := 'False'} : Bool;   // TRUE - when message prepared correctly
   END_VAR

   VAR_TEMP
      ti_MessageLength : Int;   // Message length
   END_VAR

   VAR CONSTANT
      cs_SOT : String := 'ABC';   // Message constans - SOT
      cs_EOT : String := 'XYZ';   // Message constans - EOT
      cc_Underscore : Char := '_';   // Message constans - underscore
      cc_CR : Char := '$R';   // Message constans - EOT
      cc_LF : Char := '$L';   // Message constans - EOT
   END_VAR


BEGIN
	(*
	----------------------------------------------------------------------------------------
	|                                                                                      |
	|  Copyright  2023             FORTNA Europe BV                                        |
	|  All Rights Reserved         Netherlands                                             |
	|                                                                                      |
	----------------------------------------------------------------------------------------
	Version history:
	Date        | Version   | Author       | Remark
	----------------------------------------------------------------------------------------
	27/04/2023  | 1.0       | S. Nikodem   | Release TIA 17 | DHL Munich 2023
	13/03/2024  | 1.1       | S. Nieswiec  | Added to new baseline
	*)

	REGION 1- Copy GIN

	    IF #iq_UDT_XrayInterface.Communication.SendMessage.GIN <> #si_GIN THEN

	        #si_GIN := #iq_UDT_XrayInterface.Communication.SendMessage.GIN;

	    END_IF;

	END_REGION

	REGION 2 - Prepare message

	    IF #iq_UDT_XrayInterface.Communication.SendMessage.SendTrigger
	        //AND (#si_GIN <> #si_OldGIN)             //Comment only for tests
	        AND #ix_EnableSend
	    THEN

	        //Reset Erorr
	        #s_UDT_Status.WrongMessageLength := False;

	        //Reset send message command
	        #sx_SendMessage := False;

	        //Check if previous message was sent
	        IF NOT "DB_GIN".GIN[#si_OldGIN].DHL.Xray.BagIDMessage.Sent THEN

	            "DB_GIN".GIN[#si_OldGIN].DHL.Xray.BagIDMessage.NotSent := TRUE;

	            //Only for statistics
	            #ss_Counter.MessageNotSent += 1;

	        END_IF;

	        REGION 2.1 - Copy Object ID

	            //Piece ID
	            #ss_MessageBuffer.PieceID := "DB_GIN".GIN[#si_GIN].DHL.PieceID;

	        END_REGION

	        REGION 2.2 - VID

	            //Copy VID
	            #ss_MessageBuffer.VID := "DB_GIN".GIN[#si_GIN].DHL.VID;

	        END_REGION

	        //Copy Routing Code
	        #ss_MessageBuffer.RoutingCode := "DB_GIN".GIN[#si_GIN].DHL.Xray.RoutingCode;

	        //Fill up the space to have 2 digits
	        #ti_MessageLength := LEN(#ss_MessageBuffer.RoutingCode);

	        IF #ti_MessageLength = 1 THEN
	            #ss_MessageBuffer.RoutingCode := CONCAT(IN1 := '0', IN2 := #ss_MessageBuffer.RoutingCode);
	        ELSIF #ti_MessageLength = 0 THEN
	            #ss_MessageBuffer.RoutingCode := CONCAT(IN1 := '00', IN2 := #ss_MessageBuffer.RoutingCode);
	        END_IF;

	        //Copy data from message buffer structure to String
	        //Reset variable
	        #ss_Message := '';

	        #ss_Message := CONCAT(IN1 := #cs_SOT,                        //Add SOT [ABC]
	                              IN2 := #ss_MessageBuffer.PieceID,      //Add Piece ID
	                              IN3 := #cc_Underscore,                 //Add Underscore
	                              IN4 := #ss_MessageBuffer.VID,          //Add VID
	                              IN5 := #ss_MessageBuffer.RoutingCode,  //Add Routing Code
	                              IN6 := #cs_EOT,                        //Add EOT [XYZ]
	                              IN7 := #cc_CR,                         //Add EOT [CR]
	                              IN8 := #cc_LF);                        //Add EOT [LF]

	        //Check message length
	        #ti_MessageLength := LEN(#ss_Message);

	        IF #ti_MessageLength = #i_UDT_SerialCommunicationConfiguration.SendMessageLength THEN

	            //Set varaible message is ready to send
	            #sx_SendMessage := True;

	            //Save information message is prepared to send
	            "DB_GIN".GIN[#si_GIN].DHL.Xray.BagIDMessage.MessagePrepared := True;

	            //Only for statistics
	            #ss_Counter.SendMessage += 1;

	        ELSE

	            //Set variable the message has wrong structure
	            #s_UDT_Status.WrongMessageLength := True;

	            //Save information message has wrong stucture
	            "DB_GIN".GIN[#si_GIN].DHL.Xray.BagIDMessage.WrongMessageStructure := True;

	            //Only for statisctics
	            #ss_Counter.WrongMessageLength += 1;

	        END_IF;

	        //Copy GIN
	        #si_OldGIN := #si_GIN;

	    END_IF;

	END_REGION

	REGION 3 - Send message

	    #s_Send_P2P(REQ := #sx_SendMessage
	                AND NOT #s_UDT_Status.WrongMessageLength,
	                "PORT" := #i_UDT_SerialCommunicationConfiguration."Port",
	                BUFFER := #ss_Message,
	                LENGTH := #i_UDT_SerialCommunicationConfiguration.SendMessageLength,
	                DONE => #s_UDT_Status.Done,
	                ERROR => #s_UDT_Status.Error,
	                STATUS => #s_UDT_Status.Status);

	    IF #sx_SendMessage AND #s_UDT_Status.Done THEN

	        //Reset varaible
	        #sx_SendMessage := False;

	        //Set
	        "DB_GIN".GIN[#si_GIN].DHL.Xray.BagIDMessage.Sent := True;

	        //Set Time
	        "DB_GIN".GIN[#si_GIN].DHL.Xray.BagIDMessage.SentTime := #is_ActualTime;

	        //Only for statistics
	        #ss_Counter.MessageSent += 1;

	    END_IF;

	END_REGION

	REGION 4 - Status

	    //Copy to output structure
	    #q_UDT_Status := #s_UDT_Status;

	END_REGION

END_FUNCTION_BLOCK

FUNCTION_BLOCK "FB_VFD_MultiControl_IO_Mode"
{ S7_Optimized_Access := 'TRUE' }
AUTHOR : 'KBA-PM'
VERSION : 0.1
// ATTRIBUTES
// AUTO_NUMBER = True
// BLOCK_NUMBER = 105
// END_ATTRIBUTES
   VAR_INPUT
      i_UDT_VFDConfiguration { ExternalAccessible := 'False'; ExternalVisible := 'False'; ExternalWritable := 'False'} : "UDT_VFD_MultiControl_Configuration";   //   VFD configuration structure
      i_UDT_VFDInputs { ExternalAccessible := 'False'; ExternalVisible := 'False'; ExternalWritable := 'False'} : "UDT_VFD_MultiControl_IOMode";   //   VFD inputs structure
      ii_MotorNumber { ExternalAccessible := 'False'; ExternalVisible := 'False'; ExternalWritable := 'False'} : Int;   //   Motor number that is connected to the Multicontrol module [1,2,3 or 4]
      ix_PowerOK { ExternalAccessible := 'False'; ExternalVisible := 'False'; ExternalWritable := 'False'} : Bool;   //   TRUE when External Power OK
      ix_SafetyOK { ExternalAccessible := 'False'; ExternalVisible := 'False'; ExternalWritable := 'False'} : Bool;   //   TRUE when Safety OK
      ix_SimulationModeActive { ExternalAccessible := 'False'; ExternalVisible := 'False'; ExternalWritable := 'False'} : Bool;   //   TRUE when Simulation mode active
   END_VAR

   VAR_OUTPUT
      q_UDT_HMIStatus { ExternalAccessible := 'False'; ExternalVisible := 'False'; ExternalWritable := 'False'} : "UDT_VfdStatus";   //   HMI status structure
      qsi_UDT_VFDSpeed { ExternalAccessible := 'False'; ExternalVisible := 'False'; ExternalWritable := 'False'} : SInt;   //   VFD speed setpoint
   END_VAR

   VAR_IN_OUT
      iq_UDT_ConveyorInterface : "UDT_ConveyorInterface";   //   Conveyor interface structure
      iq_UDT_VFDStatistics : "UDT_VfdStatistics";   //   Statistics structure
   END_VAR

   VAR
      s_FB_TimerOnOffDelayCheckSupply { ExternalAccessible := 'False'; ExternalVisible := 'False'; ExternalWritable := 'False'; S7_SetPoint := 'False'} : "FB_TimerOnOffDelay";   //  "TimerOnOffDelay" - to delay time for VFD supply contactor
      s_FB_TimerOnOffDelay_SafetyOK { ExternalAccessible := 'False'; ExternalVisible := 'False'; ExternalWritable := 'False'; S7_SetPoint := 'False'} : "FB_TimerOnOffDelay";   //   "TimerOnOffDelay" - to delay time for safety
      s_FB_TimerOnOffDelay_RunCommand { ExternalAccessible := 'False'; ExternalVisible := 'False'; ExternalWritable := 'False'; S7_SetPoint := 'False'} : "FB_TimerOnOffDelay";   //   "TimerOnOffDelay" - to delay time for run command motor
      s_FB_TimerOnOffDelay_PNOnline { ExternalAccessible := 'False'; ExternalVisible := 'False'; ExternalWritable := 'False'; S7_SetPoint := 'False'} : "FB_TimerOnOffDelay";
      s_R_TRIG_RunForward {InstructionName := 'R_TRIG'; LibVersion := '1.0'; ExternalAccessible := 'False'; ExternalVisible := 'False'; ExternalWritable := 'False'; S7_SetPoint := 'False'} : R_TRIG;   //   Rising edge of Run forward signal
      s_R_TRIG_RunReverse {InstructionName := 'R_TRIG'; LibVersion := '1.0'; ExternalAccessible := 'False'; ExternalVisible := 'False'; ExternalWritable := 'False'; S7_SetPoint := 'False'} : R_TRIG;   //   Rising edge of Run reverse
      s_R_TRIG_PNSlaveNotOnline {InstructionName := 'R_TRIG'; LibVersion := '1.0'; ExternalAccessible := 'False'; ExternalVisible := 'False'; ExternalWritable := 'False'; S7_SetPoint := 'False'} : R_TRIG;   //   Rising edge for trigger Profinet slave not online statistics
      s_R_TRIG_PNSlaveError {InstructionName := 'R_TRIG'; LibVersion := '1.0'; ExternalAccessible := 'False'; ExternalVisible := 'False'; ExternalWritable := 'False'; S7_SetPoint := 'False'} : R_TRIG;   //   Rising edge for trigger Profinet slave error statistics
      s_R_TRIG_InternalError {InstructionName := 'R_TRIG'; LibVersion := '1.0'; ExternalAccessible := 'False'; ExternalVisible := 'False'; ExternalWritable := 'False'; S7_SetPoint := 'False'} : R_TRIG;   //   Rising edge for trigger Internal VFD Error statistics
      s_R_TRIG_Running {InstructionName := 'R_TRIG'; LibVersion := '1.0'; ExternalAccessible := 'False'; ExternalVisible := 'False'; ExternalWritable := 'False'; S7_SetPoint := 'False'} : R_TRIG;   //   Rising edge for starting of the running signal
      s_UDT_HMIStatus { ExternalAccessible := 'False'; ExternalVisible := 'False'; ExternalWritable := 'False'; S7_SetPoint := 'False'} : "UDT_VfdStatus";   //   HMI status structure
      s_UDT_PNDevice { ExternalAccessible := 'False'; ExternalVisible := 'False'; ExternalWritable := 'False'; S7_SetPoint := 'False'} : "UDT_PNDevice";   //   PN device info structure
      ss_PNPortsStatus { ExternalAccessible := 'False'; ExternalVisible := 'False'; ExternalWritable := 'False'} : Array[1..8] of Bool;   //   TRUE when specific port has an error
      ss_VFDGeoStruct {InstructionName := 'GEOADDR'; LibVersion := '1.0'; ExternalAccessible := 'False'; ExternalVisible := 'False'; ExternalWritable := 'False'; S7_SetPoint := 'False'} : GEOADDR;   //   Geo structure indicate to telegram
      ss_RDREC { ExternalAccessible := 'False'; ExternalVisible := 'False'; ExternalWritable := 'False'} : Struct   //   Read error code record structure
         Valid { ExternalAccessible := 'False'; ExternalVisible := 'False'; ExternalWritable := 'False'} : Bool;   //      Read operation is done
         Busy { ExternalAccessible := 'False'; ExternalVisible := 'False'; ExternalWritable := 'False'} : Bool;   //      Read operation is in progress
         Error { ExternalAccessible := 'False'; ExternalVisible := 'False'; ExternalWritable := 'False'} : Bool;   //      Read operation has an error
         Status { ExternalAccessible := 'False'; ExternalVisible := 'False'; ExternalWritable := 'False'} : DWord;   //      Read operation status
         Lenght { ExternalAccessible := 'False'; ExternalVisible := 'False'; ExternalWritable := 'False'} : UInt;   //      Lenght of the read record
      END_STRUCT;
      ss_WRREC { ExternalAccessible := 'False'; ExternalVisible := 'False'; ExternalWritable := 'False'} : Struct   //   Write record structure
         Acceleration { ExternalAccessible := 'False'; ExternalVisible := 'False'; ExternalWritable := 'False'} : Struct   //      Acceleration
            REQ { ExternalAccessible := 'False'; ExternalVisible := 'False'; ExternalWritable := 'False'} : Bool;   //      Requirement
            Index { ExternalAccessible := 'False'; ExternalVisible := 'False'; ExternalWritable := 'False'} : DInt;   //      Index
            Done { ExternalAccessible := 'False'; ExternalVisible := 'False'; ExternalWritable := 'False'} : Bool;   //      Operation is done
            Busy { ExternalAccessible := 'False'; ExternalVisible := 'False'; ExternalWritable := 'False'} : Bool;   //      Write operation is in progress
            Error { ExternalAccessible := 'False'; ExternalVisible := 'False'; ExternalWritable := 'False'} : Bool;   //      Write operation has an error
            Status { ExternalAccessible := 'False'; ExternalVisible := 'False'; ExternalWritable := 'False'} : DWord;   //      Write operation status
            Data { ExternalAccessible := 'False'; ExternalVisible := 'False'; ExternalWritable := 'False'} : Word;   //      Data to write
         END_STRUCT;
         Deceleration { ExternalAccessible := 'False'; ExternalVisible := 'False'; ExternalWritable := 'False'} : Struct   //      Deceleration
            REQ { ExternalAccessible := 'False'; ExternalVisible := 'False'; ExternalWritable := 'False'} : Bool;   //      Requirement
            Index { ExternalAccessible := 'False'; ExternalVisible := 'False'; ExternalWritable := 'False'} : DInt;   //      Index
            Done { ExternalAccessible := 'False'; ExternalVisible := 'False'; ExternalWritable := 'False'} : Bool;   //      Operation is done
            Busy { ExternalAccessible := 'False'; ExternalVisible := 'False'; ExternalWritable := 'False'} : Bool;   //      Write operation is in progress
            Error { ExternalAccessible := 'False'; ExternalVisible := 'False'; ExternalWritable := 'False'} : Bool;   //      Write operation has an error
            Status { ExternalAccessible := 'False'; ExternalVisible := 'False'; ExternalWritable := 'False'} : DWord;   //      Write operation status
            Data { ExternalAccessible := 'False'; ExternalVisible := 'False'; ExternalWritable := 'False'} : Word;   //      Data to write
         END_STRUCT;
      END_STRUCT;
      s_WRREC_ACC {InstructionName := 'WRREC'; LibVersion := '1.1'; ExternalAccessible := 'False'; ExternalVisible := 'False'; ExternalWritable := 'False'; S7_SetPoint := 'False'} : WRREC;   //   Write acceleration record inctruction
      s_WRREC_DEC {InstructionName := 'WRREC'; LibVersion := '1.1'; ExternalAccessible := 'False'; ExternalVisible := 'False'; ExternalWritable := 'False'; S7_SetPoint := 'False'} : WRREC;   //   Write deceleration record instruction
      shw_VFD_Telegram { ExternalAccessible := 'False'; ExternalVisible := 'False'; ExternalWritable := 'False'} : HW_ANY;   //   Free telegram's HW_ID
      sr_MaximumSpeed { ExternalAccessible := 'False'; ExternalVisible := 'False'; ExternalWritable := 'False'} : Real;   //   Maximum speed [mm/s]
      sr_SpeedsetpointCorrected { ExternalAccessible := 'False'; ExternalVisible := 'False'; ExternalWritable := 'False'} : Real;   //  Speedsetpoint corrected with factor
      si_RequiredSpeedSetpoint { ExternalAccessible := 'False'; ExternalVisible := 'False'; ExternalWritable := 'False'} : Int;   //   Required speed setpoint
      si_AccelerationSetpoint { ExternalAccessible := 'False'; ExternalVisible := 'False'; ExternalWritable := 'False'} : Int;   //   Acceleration setpoint value
      si_DecelerationSetpoint { ExternalAccessible := 'False'; ExternalVisible := 'False'; ExternalWritable := 'False'} : Int;   //   Deceleration setpoint value
      si_AccelerationOld { ExternalAccessible := 'False'; ExternalVisible := 'False'; ExternalWritable := 'False'} : Int;   //   Old acceleration value
      si_DecelerationOld { ExternalAccessible := 'False'; ExternalVisible := 'False'; ExternalWritable := 'False'} : Int;   //   Old deceleration value
      si_ActualSpeed { ExternalAccessible := 'False'; ExternalVisible := 'False'; ExternalWritable := 'False'} : Int;   //   Actual speed in [mm/s]
      si_Log2GeoReturn { ExternalAccessible := 'False'; ExternalVisible := 'False'; ExternalWritable := 'False'} : Int;   //   Log2Geo function return
      si_Geo2LogReturn { ExternalAccessible := 'False'; ExternalVisible := 'False'; ExternalWritable := 'False'} : Int;   //   Geo2Log function return
      ssi_MotorSpeed { ExternalAccessible := 'False'; ExternalVisible := 'False'; ExternalWritable := 'False'} : SInt;   //   Motor speed value
      sx_ConfigurationError { ExternalAccessible := 'False'; ExternalVisible := 'False'; ExternalWritable := 'False'} : Bool;   //   Commissioning: configuration error
      sx_PNDeviceHealthy { ExternalAccessible := 'False'; ExternalVisible := 'False'; ExternalWritable := 'False'} : Bool;   //   Profinet device is online and error free
      sx_PowerOk { ExternalAccessible := 'False'; ExternalVisible := 'False'; ExternalWritable := 'False'} : Bool;   //   Communication, safety and power are available
      sx_VFD_Available { ExternalAccessible := 'False'; ExternalVisible := 'False'; ExternalWritable := 'False'} : Bool;   //   Hardware of VFD is ok
      sx_ErrorActive { ExternalAccessible := 'False'; ExternalVisible := 'False'; ExternalWritable := 'False'} : Bool;   //   Block has an error
      sx_InvalidMotorNumber { ExternalAccessible := 'False'; ExternalVisible := 'False'; ExternalWritable := 'False'} : Bool;   //   Invalid motor error
      sx_MotorError { ExternalAccessible := 'False'; ExternalVisible := 'False'; ExternalWritable := 'False'} : Bool;   //   Motor error
      sx_EnableOperation { ExternalAccessible := 'False'; ExternalVisible := 'False'; ExternalWritable := 'False'} : Bool;   //   Enable operation signal
      sx_RunVFDForward { ExternalAccessible := 'False'; ExternalVisible := 'False'; ExternalWritable := 'False'} : Bool;   //   Start VFD forward
      sx_RunVFDReverse { ExternalAccessible := 'False'; ExternalVisible := 'False'; ExternalWritable := 'False'} : Bool;   //   Start VFD backward
      sx_AccelerationDone { ExternalAccessible := 'False'; ExternalVisible := 'False'; ExternalWritable := 'False'} : Bool;   //   Acceleration is written
      sx_DecelerationDone { ExternalAccessible := 'False'; ExternalVisible := 'False'; ExternalWritable := 'False'} : Bool;   //   Deceleration is written
      sx_SpeedSetpointReached { ExternalAccessible := 'False'; ExternalVisible := 'False'; ExternalWritable := 'False'} : Bool;   //   Motor is running at requested speed
      sx_PNSlaveError { ExternalAccessible := 'False'; ExternalVisible := 'False'; ExternalWritable := 'False'} : Bool;   //   Profinet slave error
      sx_PNSlaveNotOnline { ExternalAccessible := 'False'; ExternalVisible := 'False'; ExternalWritable := 'False'} : Bool;   //   Profinet slave not online
      s_R_TRIG_PNSlaveNotOnline_Acyclic {InstructionName := 'R_TRIG'; LibVersion := '1.0'; ExternalAccessible := 'False'; ExternalVisible := 'False'; ExternalWritable := 'False'; S7_SetPoint := 'False'} : R_TRIG;
   END_VAR

   VAR CONSTANT
      ci_VFDArea : UInt := 1;   //   Area ID of IO Profinet devices
      ci_SubmoduleHWType : UInt := 5;   //   Submodule HW_type number
      ci_TelegramSlot : UInt := 2;   //   Free Siemens telegram slot
      ci_TelegramSubslot : UInt := 1;   //   Free Siemens telegram subslot
      cdi_ErrorCodeIndex : DInt := 17154;   //   Error code index
      cdi_AccelerationIndex : DInt := 18200;   //   Acceleration index
      cdi_DecelerationIndex : DInt := 18204;   //   Deceleration index
      ci_NumberOfProfinetPorts : Int := 2;
   END_VAR


BEGIN
	REGION Header
	(*
	----------------------------------------------------------------------------------------
	|                                                                                      |
	|  Copyright  2023             FORTNA Europe BV                                        |
	|  All Rights Reserved         Netherlands                                             |
	|                                                                                      |
	----------------------------------------------------------------------------------------

	Version history:
	Date        | Version   | Author        | Remark
	----------------------------------------------------------------------------------------
	08/11/2019  | 3.0       | A. Nowak      | Initial version
	18/03/2020  | 3.1       | K.Pokorski    | Adapting reviews
	10/06/2021  | 3.2       | L.Klar        | Region 9.1 - #ssi_MotorSpeed = 0 condition commented
	17/11/2021  | 3.3       | P.Gryszczyk   | Region 2 - RunCommand timer changed conditions
	18/02/2021  | 3.4       | P.Gryszczyk   | Region 4 - PNNotOnline and PNSlaveError masking, sending reset to system
	24/05/2023  | 3.5       | S.Nikodem     | Update to DHL Munich specification
	07/06/2023  | 3.6       | R.Golonka     | Update to new UDT_VFD_Multicontrol_IOMode, Hardware IO Mode module changed
	04/07/2023  | 3.7       | P.Gryszczyk   | Changed the PNSlaveNotOnline to R_TRIG for the acyclic writing logic
	08/08/2023  | 3.8       | R.Golonka     | Adjust alarm the device, Added profinet slave warning
	30/08/2023  | 4.0       | S.Theocharis  | Mask pn error when not online is set
	13/03/2024  | 4.1       | S. Nieswiec   | Added to new baseline
	*)
	END_REGION

	REGION 1 - Get Device Profinet number

	    // Getting information about Profinet device
	    "FC_GetDevicePN"(is_PNDeviceName := #i_UDT_VFDConfiguration.VFDPNDeviceName,
	                     ix_SimulationModeActive := #ix_SimulationModeActive,
	                     iqUDT_PND := #s_UDT_PNDevice);

	    // Getting information about port status of device
	    "FC_GetPNPortStatus"(ii_NumberOfPorts := #ci_NumberOfProfinetPorts,
	                         iUDT_DevicePNInfo := #s_UDT_PNDevice,
	                         qa_PortFault => #ss_PNPortsStatus);

	END_REGION

	REGION 2 - Motor number validation

	    // Check the motor number and copy the it's error status and speed.
	    CASE (#ii_MotorNumber)
	    OF
	        1:
	            // Delay
	            #s_FB_TimerOnOffDelay_RunCommand(iudi_OnDelayTime := 1500,
	                                             ix_SignalToDelay := #sx_RunVFDForward OR #sx_RunVFDReverse);

	            #ssi_MotorSpeed := #i_UDT_VFDInputs.SpeedMotor1;

	            #sx_MotorError := #i_UDT_VFDInputs.ErrorMotor1;

	        2:
	            #s_FB_TimerOnOffDelay_RunCommand(iudi_OnDelayTime := 1500,
	                                             ix_SignalToDelay := #sx_RunVFDForward OR #sx_RunVFDReverse);

	            #ssi_MotorSpeed := #i_UDT_VFDInputs.SpeedMotor2;

	            #sx_MotorError := #i_UDT_VFDInputs.ErrorMotor2;
	        3:
	            #s_FB_TimerOnOffDelay_RunCommand(iudi_OnDelayTime := 1500,
	                                             ix_SignalToDelay := #sx_RunVFDForward OR #sx_RunVFDReverse);

	            #ssi_MotorSpeed := #i_UDT_VFDInputs.SpeedMotor3;

	            #sx_MotorError := #i_UDT_VFDInputs.ErrorMotor3;
	        4:
	            #s_FB_TimerOnOffDelay_RunCommand(iudi_OnDelayTime := 1500,
	                                             ix_SignalToDelay := #sx_RunVFDForward OR #sx_RunVFDReverse);

	            #ssi_MotorSpeed := #i_UDT_VFDInputs.SpeedMotor4;

	            #sx_MotorError := #i_UDT_VFDInputs.ErrorMotor4;

	        ELSE
	            #sx_InvalidMotorNumber := TRUE;
	    END_CASE;

	END_REGION

	REGION 3 - Reset errors

	    // Reset the errors on the command from the conveyor interface.
	    IF #iq_UDT_ConveyorInterface.InternalErrorReset OR (NOT #iq_UDT_ConveyorInterface.HardwareOk AND #s_UDT_HMIStatus.PNSlaveNotonline) THEN
	        #s_UDT_HMIStatus.PNSlaveNotonline := FALSE;
	        #s_UDT_HMIStatus.PNSlaveError := FALSE;
	        #s_UDT_HMIStatus.InternalError := FALSE;
	        #s_UDT_HMIStatus.PNSlaveWarning := FALSE;
	        #sx_PNSlaveError := FALSE;
	        #sx_PNSlaveNotOnline := FALSE;
	        #sx_InvalidMotorNumber := FALSE;
	        #sx_MotorError := FALSE;
	    END_IF;

	END_REGION

	REGION 4 - Hardware check

	    // Hardware will be available only after the delay, so the device has time for the initialization.
	    #s_FB_TimerOnOffDelayCheckSupply(iudi_OnDelayTime := 2000,
	                                     ix_SignalToDelay := #ix_PowerOK,
	                                     qx_DelayedSignal => #sx_PowerOk);

	    IF NOT "DB_ProfinetDiagnostic".ProfinetNetworks[#s_UDT_PNDevice.PNNetworknumber].DeviceStatus[#s_UDT_PNDevice.PNDeviceNumber].DeviceState.Exist
	        AND NOT #ix_SimulationModeActive
	        AND #sx_PowerOk
	        AND #iq_UDT_ConveyorInterface.HardwareOk
	    THEN
	        #sx_PNSlaveNotOnline := True;
	    END_IF;

	    // Chceck if PN ports are healthy
	    IF #ss_PNPortsStatus[1] XOR #ss_PNPortsStatus[2] THEN
	        #s_UDT_HMIStatus.PNSlaveWarning := TRUE;
	    END_IF;

	    // Check if PN device has an error
	    IF "DB_ProfinetDiagnostic".ProfinetNetworks[#s_UDT_PNDevice.PNNetworknumber].DeviceStatus[#s_UDT_PNDevice.PNDeviceNumber].DeviceState.Error
	        AND NOT #ix_SimulationModeActive
	        AND #sx_PowerOk
	        AND NOT #s_UDT_HMIStatus.PNSlaveWarning
	        AND #iq_UDT_ConveyorInterface.HardwareOk
	        AND NOT #sx_PNSlaveNotOnline
	    THEN
	        #sx_PNSlaveError := TRUE;
	    END_IF;

	    // Set bit when PN device is healthy (online and no error)
	    #sx_PNDeviceHealthy :=
	    NOT #s_UDT_HMIStatus.PNSlaveNotonline
	    AND NOT #s_UDT_HMIStatus.PNSlaveError
	    AND #s_UDT_PNDevice.PNDeviceFound
	    AND #sx_PowerOk;

	    // Set VFD available bit when all conditions are met.
	    #sx_VFD_Available :=
	    (NOT #sx_MotorError
	    AND #sx_PowerOk
	    AND #sx_PNDeviceHealthy)
	    OR #ix_SimulationModeActive;

	END_REGION

	REGION 5 - Extract telegram's HW_ID

	    // Extract telegram's HW_ID //Do we need this in every scan?
	    #si_Log2GeoReturn := LOG2GEO(LADDR := "DB_ProfinetDiagnostic".ProfinetNetworks[#s_UDT_PNDevice.PNNetworknumber].DeviceStatus[#s_UDT_PNDevice.PNDeviceNumber].DeviceState.HW_ID, GEOADDR := #ss_VFDGeoStruct);
	    #ss_VFDGeoStruct.AREA := #ci_VFDArea;
	    #ss_VFDGeoStruct.HWTYPE := #ci_SubmoduleHWType;
	    #ss_VFDGeoStruct.STATION := INT_TO_UINT(#s_UDT_PNDevice.PNDeviceNumber);
	    #ss_VFDGeoStruct.SLOT := #ci_TelegramSlot;
	    #ss_VFDGeoStruct.SUBSLOT := #ci_TelegramSubslot;

	    #si_Geo2LogReturn := GEO2LOG(GEOADDR := #ss_VFDGeoStruct, LADDR => #shw_VFD_Telegram);

	END_REGION

	REGION 6 - Check errors

	    #s_FB_TimerOnOffDelay_SafetyOK(iudi_OnDelayTime := 10000,
	                                   ix_SignalToDelay := #ix_SafetyOK);

	    #s_FB_TimerOnOffDelay_PNOnline(iudi_OnDelayTime := 4000,
	                                   ix_SignalToDelay := "DB_ProfinetDiagnostic".ProfinetNetworks[#s_UDT_PNDevice.PNNetworknumber].DeviceStatus[#s_UDT_PNDevice.PNDeviceNumber].DeviceState.Exist);


	    // Check if the motor has an error.
	    IF #sx_MotorError
	        /// OR(#i_UDT_VFDInputs.Error = 3)) // Remvoved the global error to focus on the individual roller
	        AND #s_FB_TimerOnOffDelay_SafetyOK.qx_DelayedSignal
	        AND #s_FB_TimerOnOffDelay_PNOnline.qx_DelayedSignal
	        AND #sx_PowerOk
	    THEN
	        #s_UDT_HMIStatus.InternalError := TRUE;
	    END_IF;

	    #s_R_TRIG_InternalError(CLK := #s_UDT_HMIStatus.InternalError);

	    // If there is an internal error, read the error code from the Interroll VFD. Otherwise, reset it.
	    IF #s_R_TRIG_InternalError.Q THEN
	        #s_UDT_HMIStatus.ErrorCode := #i_UDT_VFDInputs.LastError;
	    END_IF;

	    //Reset Error code
	    IF NOT #s_UDT_HMIStatus.InternalError THEN
	        #s_UDT_HMIStatus.ErrorCode := 0;
	    END_IF;

	END_REGION

	REGION 7 - Check if configuration is ok for commissioning purposes

	    // Validate the VFD configuration and motor number.
	    IF #i_UDT_VFDConfiguration.MaximumSpeed > 0.0
	        AND #i_UDT_VFDConfiguration.VFDRampUpTime > 0
	        AND #i_UDT_VFDConfiguration.VFDRampDownTime > 0
	        AND NOT #sx_InvalidMotorNumber
	    THEN
	        #sx_ConfigurationError := FALSE;
	    ELSE
	        #sx_ConfigurationError := TRUE;
	    END_IF;

	END_REGION

	REGION 8 - Handle speed

	    // Write max speed to static.
	    #sr_MaximumSpeed := #i_UDT_VFDConfiguration.MaximumSpeed;

	    // Use correction factor to calculate setpint for diaginal use
	    #sr_SpeedsetpointCorrected := INT_TO_REAL(#iq_UDT_ConveyorInterface.SpeedSetpoint) * #i_UDT_VFDConfiguration.CorrectionFactor;

	    // Actual speed setpoint
	    #si_RequiredSpeedSetpoint := REAL_TO_INT((#sr_SpeedsetpointCorrected * 100.0) / (#sr_MaximumSpeed));

	    // Speed setpoint saturation in case when the speed setpoint is higher than the max speed.
	    IF #si_RequiredSpeedSetpoint > 100
	    THEN
	        #si_RequiredSpeedSetpoint := 100;
	        #iq_UDT_ConveyorInterface.ConfigurationError := TRUE;
	    ELSIF #si_RequiredSpeedSetpoint < -100
	    THEN
	        #si_RequiredSpeedSetpoint := -100;
	        #iq_UDT_ConveyorInterface.ConfigurationError := TRUE;
	    END_IF;
	END_REGION

	REGION 9 - Prepare output data VFD

	    REGION 9.1 - Set speed setpoint in forward and reverse direction
	        // Get rising edge of Run forward and reverse signal.
	        #s_R_TRIG_RunForward(CLK := #iq_UDT_ConveyorInterface.RunFwd);
	        #s_R_TRIG_RunReverse(CLK := #iq_UDT_ConveyorInterface.RunRvs);

	        // When rising edge of the forward or reverse signal is received, the drive has to stop to be able to make the switch.
	        IF #s_R_TRIG_RunForward.Q
	            OR #s_R_TRIG_RunReverse.Q
	        THEN
	            #qsi_UDT_VFDSpeed := 0;
	        END_IF;

	        // If motor stopped and Run forward is requested and forward direction is interlock, set run forward signal and reset run reverse signal.
	        IF //#ssi_MotorSpeed = 0 and
	            #iq_UDT_ConveyorInterface.RunFwd
	            AND #i_UDT_VFDConfiguration.InterlockFwd
	        THEN
	            #sx_RunVFDForward := TRUE;
	            #sx_RunVFDReverse := FALSE;
	        END_IF;

	        // If motor stopped and Run reverse is requested and reverse direction is interlock, set run reverse signal and reset run forward signal.
	        IF // #ssi_MotorSpeed = 0 AND
	            #iq_UDT_ConveyorInterface.RunRvs
	            AND #i_UDT_VFDConfiguration.InterlockRvs
	        THEN
	            #sx_RunVFDReverse := TRUE;
	            #sx_RunVFDForward := FALSE;
	        END_IF;

	    END_REGION

	    REGION 9.2 - Stopping

	        // Stop the VFD if one of the following conditions is met.
	        IF (NOT #iq_UDT_ConveyorInterface.RunRvs AND NOT #iq_UDT_ConveyorInterface.RunFwd)
	            OR (#iq_UDT_ConveyorInterface.RunRvs AND #iq_UDT_ConveyorInterface.RunFwd)
	            OR (#sx_RunVFDReverse AND NOT #i_UDT_VFDConfiguration.InterlockRvs)
	            OR (#sx_RunVFDForward AND NOT #i_UDT_VFDConfiguration.InterlockFwd)
	            OR ((#s_R_TRIG_RunForward.Q AND #ssi_MotorSpeed < 0)
	            OR (#s_R_TRIG_RunReverse.Q AND #ssi_MotorSpeed > 0))
	        THEN
	            #sx_RunVFDReverse := FALSE;
	            #sx_RunVFDForward := FALSE;
	        END_IF;

	    END_REGION

	    REGION 9.3 - Check for enable operation signal

	        // Operation is enable when VFD is available and there is one of the run commands.
	        #sx_EnableOperation :=
	        #sx_VFD_Available
	        AND (#sx_RunVFDForward OR #sx_RunVFDReverse)
	        AND NOT #sx_ConfigurationError;

	    END_REGION

	END_REGION

	REGION 10 - Write outputs to VFD

	    REGION 10.1 - Write speed setpoint to drive

	        // The conveyor stopped and may now run in forward direction.
	        IF ((#sx_RunVFDForward AND NOT #i_UDT_VFDConfiguration.DirectionReversal)
	            OR (#sx_RunVFDReverse AND #i_UDT_VFDConfiguration.DirectionReversal))
	            AND #sx_EnableOperation
	        THEN
	            #qsi_UDT_VFDSpeed := INT_TO_SINT(#si_RequiredSpeedSetpoint);
	        END_IF;

	        // The conveyor stopped and may now run in reverse direction.
	        IF ((#sx_RunVFDReverse AND NOT #i_UDT_VFDConfiguration.DirectionReversal)
	            OR (#sx_RunVFDForward AND #i_UDT_VFDConfiguration.DirectionReversal))
	            AND #sx_EnableOperation
	        THEN
	            #qsi_UDT_VFDSpeed := - INT_TO_SINT(#si_RequiredSpeedSetpoint);
	        END_IF;

	        // Clear speed setpoint when run isn't request.
	        IF (NOT #sx_RunVFDForward
	            AND NOT #sx_RunVFDReverse)
	            OR NOT #sx_EnableOperation
	        THEN
	            #qsi_UDT_VFDSpeed := 0;
	        END_IF;

	    END_REGION

	    REGION 10.2 - Calculate acceleration and deceleration values

	        // Recalculating Acceleration ramp - deviding maximum configured speed by Ramp up time and devide it by 1000.
	        #si_AccelerationSetpoint := REAL_TO_INT(#sr_MaximumSpeed / (UDINT_TO_REAL(#i_UDT_VFDConfiguration.VFDRampUpTime) / 1000.0));

	        // Recalculating Deceleration ramp - deviding maximum configured speed by Ramp down time and devide it by 1000.
	        #si_DecelerationSetpoint := REAL_TO_INT(#sr_MaximumSpeed / (UDINT_TO_REAL(#i_UDT_VFDConfiguration.VFDRampDownTime) / 1000.0));

	    END_REGION

	    REGION 10.3 - Write acceleration to drive

	        #s_R_TRIG_PNSlaveNotOnline_Acyclic(CLK := NOT #s_UDT_HMIStatus.PNSlaveNotonline);


	        // Acceleration write operation is done.
	        IF #sx_AccelerationDone
	        THEN
	            // There is new acceleration value or device is offline.
	            IF #si_AccelerationSetpoint <> #si_AccelerationOld
	                OR #s_R_TRIG_PNSlaveNotOnline_Acyclic.Q
	            THEN
	                // Reset the accleration operation done signal.
	                #sx_AccelerationDone := FALSE;
	            END_IF;
	        END_IF;

	        // The acceleration operation isn't done or there is first scan and device is online.
	        IF (NOT #sx_AccelerationDone OR "mx_FirstScan")
	            AND NOT #s_UDT_HMIStatus.PNSlaveNotonline
	        THEN

	            // There isn't an invalid motor number error and acceleration isn't equal to 0.
	            IF NOT #sx_InvalidMotorNumber
	                AND #si_AccelerationSetpoint > 0
	            THEN
	                // Calculate the index of the acceleration.
	                #ss_WRREC.Acceleration.Index := #cdi_AccelerationIndex + #ii_MotorNumber;
	                // Prepare the data.
	                #ss_WRREC.Acceleration.Data := SWAP(INT_TO_WORD(#si_AccelerationSetpoint));
	                // Set operation is required.
	                #ss_WRREC.Acceleration.REQ := TRUE;

	                // Send acceleration to the device.
	                #s_WRREC_ACC(REQ := #ss_WRREC.Acceleration.REQ,
	                             ID := #shw_VFD_Telegram,
	                             INDEX := #ss_WRREC.Acceleration.Index,
	                             LEN := 0,
	                             DONE => #ss_WRREC.Acceleration.Done,
	                             BUSY => #ss_WRREC.Acceleration.Busy,
	                             ERROR => #ss_WRREC.Acceleration.Error,
	                             STATUS => #ss_WRREC.Acceleration.Status,
	                             RECORD := #ss_WRREC.Acceleration.Data);

	                // Send operation is done.
	                IF #ss_WRREC.Acceleration.Done
	                THEN
	                    // Reset operation is required bit.
	                    #ss_WRREC.Acceleration.REQ := FALSE;
	                    // Set the operation is done signal.
	                    #sx_AccelerationDone := TRUE;
	                    // Write acceleration value into the old one.
	                    #si_AccelerationOld := #si_AccelerationSetpoint;
	                END_IF;
	            END_IF;
	        END_IF;

	    END_REGION

	    REGION 10.4 - Write deceleration to drive

	        // Deceleration write operation is done.
	        IF #sx_DecelerationDone
	        THEN
	            // There is new deceleration value or device is offline.
	            IF #si_DecelerationSetpoint <> #si_DecelerationOld
	                OR #s_R_TRIG_PNSlaveNotOnline_Acyclic.Q
	            THEN
	                // Reset the deceleration operation done signal.
	                #sx_DecelerationDone := FALSE;
	            END_IF;
	        END_IF;

	        // The deceleration operation isn't done or there is first scan and device is online.
	        IF (NOT #sx_DecelerationDone OR "mx_FirstScan")
	            AND NOT #s_UDT_HMIStatus.PNSlaveNotonline
	        THEN
	            // There isn't an invalid motor number error and deceleration isn't equal to 0.
	            IF NOT #sx_InvalidMotorNumber
	                AND #si_DecelerationSetpoint > 0
	            THEN
	                // Calculate the index of the deceleration.
	                #ss_WRREC.Deceleration.Index := #cdi_DecelerationIndex + #ii_MotorNumber;
	                // Prepare the data.
	                #ss_WRREC.Deceleration.Data := SWAP(INT_TO_WORD(#si_DecelerationSetpoint));
	                // Set operation is required.
	                #ss_WRREC.Deceleration.REQ := TRUE;

	                // Send deceleration to the device.
	                #s_WRREC_DEC(REQ := #ss_WRREC.Deceleration.REQ,
	                             ID := #shw_VFD_Telegram,
	                             INDEX := #ss_WRREC.Deceleration.Index,
	                             LEN := 0,
	                             DONE => #ss_WRREC.Deceleration.Done,
	                             BUSY => #ss_WRREC.Deceleration.Busy,
	                             ERROR => #ss_WRREC.Deceleration.Error,
	                             STATUS => #ss_WRREC.Deceleration.Status,
	                             RECORD := #ss_WRREC.Deceleration.Data);

	                // Send operation is done.
	                IF #ss_WRREC.Deceleration.Done
	                THEN
	                    // Reset operation is required bit.
	                    #ss_WRREC.Deceleration.REQ := FALSE;
	                    // Set the operation is done signal.
	                    #sx_DecelerationDone := TRUE;
	                    // Write deceleration value into the old one.
	                    #si_DecelerationOld := #si_DecelerationSetpoint;
	                END_IF;
	            END_IF;
	        END_IF;

	    END_REGION

	END_REGION

	REGION 11 - Copy signals to interface DB and to status output UDT

	    // Create collective error.
	    #sx_ErrorActive :=
	    #s_UDT_HMIStatus.PNSlaveNotonline
	    OR #s_UDT_HMIStatus.PNSlaveError
	    OR #s_UDT_HMIStatus.InternalError
	    OR #sx_ConfigurationError;

	    // Motor is giving direct signal on start, move setpoint to actual speed.
	    IF #ssi_MotorSpeed > 0
	    THEN
	        #si_ActualSpeed := #iq_UDT_ConveyorInterface.SpeedSetpoint;
	        #sx_SpeedSetpointReached := TRUE;
	    ELSIF #ssi_MotorSpeed < 0
	    THEN
	        #si_ActualSpeed := (-1) * #iq_UDT_ConveyorInterface.SpeedSetpoint;
	        #sx_SpeedSetpointReached := TRUE;
	    ELSE
	        #si_ActualSpeed := 0;
	        #sx_SpeedSetpointReached := FALSE;
	    END_IF;

	    //For direction reversal negate the actual speed
	    IF #i_UDT_VFDConfiguration.DirectionReversal THEN
	        #si_ActualSpeed := (-1) * #si_ActualSpeed;
	    END_IF;


	    // Write interface bits.
	    #iq_UDT_ConveyorInterface.VFDRunning :=
	    #sx_VFD_Available
	    AND #iq_UDT_ConveyorInterface.ActualSpeed <> 0;

	    // Speed setpoint is reached.
	    #iq_UDT_ConveyorInterface.VFDatSpeed :=
	    #sx_SpeedSetpointReached
	    AND #sx_VFD_Available;

	    // Set the internal VFD error bit if any fault is active.
	    #iq_UDT_ConveyorInterface.InternalErrorVFD := #sx_ErrorActive;
	    // Copy the speed value to the output.

	    #iq_UDT_ConveyorInterface.ActualSpeed := #si_ActualSpeed;

	    //Copy error PN slave not online status to HMI status
	    #s_UDT_HMIStatus.PNSlaveNotonline := #sx_PNSlaveNotOnline;
	    //Copy error PN slave status to HMI status
	    #s_UDT_HMIStatus.PNSlaveError := #sx_PNSlaveError;

	    // Copy error status to output.
	    #q_UDT_HMIStatus := #s_UDT_HMIStatus;

	END_REGION

	REGION 12 - Statistics

	    // Create trigger on error and create statistics for profinet slave not online.
	    #s_R_TRIG_PNSlaveNotOnline(CLK := #s_UDT_HMIStatus.PNSlaveNotonline);

	    IF #iq_UDT_ConveyorInterface.ResetStatistics
	        OR #s_UDT_HMIStatus.PNSlaveNotonline
	    THEN
	        "FC_Statistics"(ix_Reset := #iq_UDT_ConveyorInterface.ResetStatistics,
	                        ix_Activate := #s_UDT_HMIStatus.PNSlaveNotonline,
	                        ix_RTrigActivate := #s_R_TRIG_PNSlaveNotOnline.Q,
	                        iqUDT_Statistics := #iq_UDT_VFDStatistics.PNSlaveNotOnline);
	    END_IF;

	    // Create trigger on error and create statistics for profinet slave error.
	    #s_R_TRIG_PNSlaveError(CLK := #s_UDT_HMIStatus.PNSlaveError);

	    IF #iq_UDT_ConveyorInterface.ResetStatistics
	        OR #s_UDT_HMIStatus.PNSlaveError
	    THEN
	        "FC_Statistics"(ix_Reset := #iq_UDT_ConveyorInterface.ResetStatistics,
	                        ix_Activate := #s_UDT_HMIStatus.PNSlaveError,
	                        ix_RTrigActivate := #s_R_TRIG_PNSlaveError.Q,
	                        iqUDT_Statistics := #iq_UDT_VFDStatistics.PNSlaveError);
	    END_IF;

	    IF #iq_UDT_ConveyorInterface.ResetStatistics
	        OR #s_UDT_HMIStatus.InternalError
	    THEN
	        "FC_Statistics"(ix_Reset := #iq_UDT_ConveyorInterface.ResetStatistics,
	                        ix_Activate := #s_UDT_HMIStatus.InternalError,
	                        ix_RTrigActivate := #s_R_TRIG_InternalError.Q,
	                        iqUDT_Statistics := #iq_UDT_VFDStatistics.VFDInternalError);
	    END_IF;

	    // Create trigger on running signal and create statistics for running status.
	    #s_R_TRIG_Running(CLK := #iq_UDT_ConveyorInterface.VFDRunning);

	    IF #iq_UDT_ConveyorInterface.ResetStatistics
	        OR #iq_UDT_ConveyorInterface.VFDRunning
	    THEN
	        "FC_Statistics"(ix_Reset := #iq_UDT_ConveyorInterface.ResetStatistics,
	                        ix_Activate := #iq_UDT_ConveyorInterface.VFDRunning,
	                        ix_RTrigActivate := #s_R_TRIG_Running.Q,
	                        iqUDT_Statistics := #iq_UDT_VFDStatistics.Running);
	    END_IF;

	END_REGION
END_FUNCTION_BLOCK

FUNCTION_BLOCK "FB_TrackingMonitor"
{ S7_Optimized_Access := 'TRUE' }
VERSION : 0.1
// ATTRIBUTES
// AUTO_NUMBER = True
// BLOCK_NUMBER = 104
// END_ATTRIBUTES
   VAR_INPUT
      ix_Enable { ExternalAccessible := 'False'; ExternalVisible := 'False'; ExternalWritable := 'False'} : Bool;   // One Shot or Constant TRUE to exectue
      ii_StartPointer { ExternalAccessible := 'False'; ExternalVisible := 'False'; ExternalWritable := 'False'} : Int;
      ii_EndPointer { ExternalAccessible := 'False'; ExternalVisible := 'False'; ExternalWritable := 'False'} : Int;
      i_UDT_ConveyorCommonConfiguration { ExternalAccessible := 'False'; ExternalVisible := 'False'; ExternalWritable := 'False'} : "UDT_ConveyorCommonConfiguration";   // Conveyor common configuration
   END_VAR

   VAR_OUTPUT
      qx_ErrorCode { ExternalAccessible := 'False'; ExternalVisible := 'False'; ExternalWritable := 'False'} : Int;
      q_Overview { ExternalAccessible := 'False'; ExternalVisible := 'False'; ExternalWritable := 'False'} : "UDT_TrackingOverview";
   END_VAR

   VAR_IN_OUT
      iq_Object : Array[*] of "UDT_TrackingMonitor";
      iq_Tracking : Array[*] of Int;
   END_VAR

   VAR
      sdi_TotalConvLength { ExternalAccessible := 'False'; ExternalVisible := 'False'; ExternalWritable := 'False'} : DInt;
      si_StartPointer { ExternalAccessible := 'False'; ExternalVisible := 'False'; ExternalWritable := 'False'} : Int;
      si_EndPointer { ExternalAccessible := 'False'; ExternalVisible := 'False'; ExternalWritable := 'False'} : Int;
      si_NextObject { ExternalAccessible := 'False'; ExternalVisible := 'False'; ExternalWritable := 'False'} : Int;
      si_FirstObject { ExternalAccessible := 'False'; ExternalVisible := 'False'; ExternalWritable := 'False'} : Int;
      si_LengthOfMonitoringArray { ExternalAccessible := 'False'; ExternalVisible := 'False'; ExternalWritable := 'False'} : UInt;
      si_PreviousID { ExternalAccessible := 'False'; ExternalVisible := 'False'; ExternalWritable := 'False'} : Int;
   END_VAR

   VAR_TEMP
      ti_index : Int;
      ret_val : Int;
      t_udt_TrackingMonitor : "UDT_TrackingMonitor";
      ti_fill : Int;
   END_VAR


BEGIN
	(*
	----------------------------------------------------------------------------------------
	|                                                                                      |
	|                              FORTNA Europe                                           |
	|                              Netherlands                                             |
	|                                                                                      |
	----------------------------------------------------------------------------------------

	Version history:
	Date        | Version   | Author            | Remark
	----------------------------------------------------------------------------------------
	05/05/2023  | 0.1       | S. Theocharis     | first release
	13/03/2024  | 1.1       | S. Nieswiec       | Added to new baseline
	*)

	REGION 1 Check Condition to execute

	    IF NOT #ix_Enable THEN
	        RETURN;
	    END_IF;

	END_REGION

	REGION 2 Initialize variables

	    //Clear value
	    #ti_fill := 0;

	    //Reset Error
	    #qx_ErrorCode := 0;

	    //Clear UDT
	    #t_udt_TrackingMonitor.Data := 0;
	    #t_udt_TrackingMonitor.Position := 0;

	    // Check the conveyor length
	    #sdi_TotalConvLength := (#i_UDT_ConveyorCommonConfiguration.Length + #i_UDT_ConveyorCommonConfiguration.LengthCorrection) / 10;


	    //Define start of  search window
	    IF #ii_StartPointer > 0 THEN
	        #si_StartPointer := #ii_StartPointer;
	    ELSE
	        #si_StartPointer := 0;
	    END_IF;

	    //Define end of search window
	    IF (#ii_EndPointer > 0) AND (#ii_EndPointer > #si_StartPointer) THEN
	        #si_EndPointer := #ii_EndPointer;
	    ELSE
	        #si_EndPointer := DINT_TO_INT(#sdi_TotalConvLength);
	    END_IF;


	    //Verifiy pointers
	    IF #si_EndPointer <= #si_StartPointer THEN
	        #qx_ErrorCode := 2;
	        RETURN; //exit block
	    END_IF;


	    //Check length of monitoring array
	    #si_LengthOfMonitoringArray := INT_TO_UINT("FC_GetNrOfArrayEl"(#iq_Object));
	    #si_NextObject := DINT_TO_INT(LOWER_BOUND(ARR := #iq_Object, DIM := 1));
	    #si_FirstObject := #si_NextObject;
	    //make dynamic the length of the tracking monitor DB
	    //clear tracking monitor
	    #ret_val := MOVE_BLK_VARIANT(SRC := #t_udt_TrackingMonitor, COUNT := #si_LengthOfMonitoringArray, SRC_INDEX := 0, DEST_INDEX := #si_NextObject, DEST => #iq_Object);

	END_REGION

	REGION 3 Reb-build tracking monitor
	    (* do we distinguish parcel from window? *)

	    FOR #ti_index := #si_StartPointer TO #si_EndPointer BY 1 DO

	        IF #iq_Tracking[#ti_index] <> 0
	            AND #iq_Tracking[#ti_index] <> #si_PreviousID  //in case we have multiple entires with the same GIN or Data
	        THEN
	            #iq_Object[#si_NextObject].Data := #iq_Tracking[#ti_index];  //Copy Data to onbect ID
	            #iq_Object[#si_NextObject].Position := #ti_index;
	            #iq_Object[#si_NextObject].DataLength := 1;

	            #si_NextObject += 1; //increment for next cycle

	            //Overflow handling
	            IF #si_NextObject >= #si_LengthOfMonitoringArray THEN
	                #qx_ErrorCode := 1;  // 1 = more then 30 objects detected
	                #si_NextObject := DINT_TO_INT(LOWER_BOUND(ARR := #iq_Object, DIM := 1));
	                EXIT;
	            END_IF;


	        ELSIF (#iq_Tracking[#ti_index] = #si_PreviousID)
	            AND #si_PreviousID <> 0
	        THEN

	            //Increment Data lentgh
	            #iq_Object[#si_NextObject - 1].DataLength += 1;

	        END_IF;

	        //save ID for next loop
	        #si_PreviousID := #iq_Tracking[#ti_index];

	    END_FOR;

	    //Clear empty positions
	    FOR #ti_index := #si_NextObject TO DINT_TO_INT(UPPER_BOUND(ARR := #iq_Object, DIM := 1)) BY 1 DO
	        #iq_Object[#ti_index].Data := 0;
	        #iq_Object[#ti_index].Position := 0;
	        #iq_Object[#ti_index].DataLength := 0;
	    END_FOR;



	END_REGION

	REGION Tracking overwiev

	    //Count lenght from all detected parcel
	    FOR #ti_index := 1 TO #si_NextObject BY 1 DO

	        #ti_fill := #ti_fill + #iq_Object[#ti_index].DataLength;

	    END_FOR;

	    //Rewwrite dates on output
	    #q_Overview.TotalObject := #si_NextObject - 1;
	    #q_Overview.FillingRate := REAL_TO_INT((INT_TO_REAL(#ti_fill) / (INT_TO_REAL(#si_EndPointer - #ii_StartPointer))) * 100.0);


	END_REGION

END_FUNCTION_BLOCK

FUNCTION_BLOCK "FB_CheckParcelData"
{ S7_Optimized_Access := 'TRUE' }
VERSION : 0.1
// ATTRIBUTES
// AUTO_NUMBER = True
// BLOCK_NUMBER = 239
// END_ATTRIBUTES
   VAR_INPUT
      ii_GIN { ExternalAccessible := 'False'; ExternalVisible := 'False'; ExternalWritable := 'False'} : Int;   // GIN number
      ii_XrayLocation { ExternalAccessible := 'False'; ExternalVisible := 'False'; ExternalWritable := 'False'} : Int;   // X-ray location
      ii_SourceNode { ExternalAccessible := 'False'; ExternalVisible := 'False'; ExternalWritable := 'False'} : Int;   // ID Source Node
      ii_DestinationNode { ExternalAccessible := 'False'; ExternalVisible := 'False'; ExternalWritable := 'False'} : Int;   // ID Destination Node
      is_ActualTime { ExternalAccessible := 'False'; ExternalVisible := 'False'; ExternalWritable := 'False'} : String;   // Actual date annd time in String
   END_VAR

   VAR_IN_OUT
      iq_UDT_FifoHeader : "UDT_FifoHeader";   // FIFO header
      iqa_FifoData : Array[*] of "UDT_MessageV2";   // FIFO data buffer
      iqi_MessageSequenceNumber { ExternalAccessible := 'False'; ExternalVisible := 'False'; ExternalWritable := 'False'} : Int;   // Message number
   END_VAR

   VAR
      FB_MFC_Sort_COY_ReceiveResult_Instance { ExternalAccessible := 'False'; ExternalVisible := 'False'; ExternalWritable := 'False'; S7_SetPoint := 'False'} : "FB_MFC_Sort_COY_ReceiveResult";
      PieceID { ExternalAccessible := 'False'; ExternalVisible := 'False'; ExternalWritable := 'False'} : String[40];
   END_VAR

   VAR_TEMP
      ts_String : String;
   END_VAR


BEGIN
	(*
	----------------------------------------------------------------------------------------
	|                                                                                      |
	|  Copyright  2023             FORTNA Europe BV                                        |
	|  All Rights Reserved         Netherlands                                             |
	|                                                                                      |
	----------------------------------------------------------------------------------------
	Version history:
	Date        | Version   | Author       | Remark
	----------------------------------------------------------------------------------------
	05/10/2023  | 1.0       | S. Nikodem   | Release TIA 17 | DHL Munich 2023
	12/03/2024  | 1.1       | S. Nieswiec  | Added to new Baseline
	*)

	REGION Check Piece ID

	    IF #ii_GIN > 0 THEN

	        IF "DB_GIN".GIN[#ii_GIN].DHL.PieceID = '' THEN

	            //Generation Piece ID
	            //Constant
	            #PieceID[1] := '0';
	            #PieceID[2] := '0';
	            #PieceID[3] := '0';
	            #PieceID[4] := '0';
	            #PieceID[5] := '0';
	            #PieceID[6] := '0';
	            #PieceID[7] := '0';
	            #PieceID[8] := '_';
	            #PieceID[9] := 'L';
	            #PieceID[10] := 'O';
	            #PieceID[11] := 'S';
	            #PieceID[12] := 'T';
	            #PieceID[13] := '_';
	            #PieceID[14] := 'X';
	            #PieceID[15] := 'R';
	            #PieceID[16] := 'A';
	            #PieceID[17] := 'Y';
	            #PieceID[18] := '_';

	            //XrayLocation
	            #ts_String := DELETE(IN := DINT_TO_STRING(#ii_XrayLocation), L := 1, P := 1);
	            #PieceID[19] := #ts_String[1];
	            #PieceID[20] := #ts_String[2];
	            #PieceID[21] := #ts_String[3];

	            //Constant
	            #PieceID[22] := '_';

